C05398=1044.038,401.333,-130.987,174.157,43.481,158.582
C05399=1044.028,401.087,-130.943,174.149,43.474,158.580
C05400=1044.019,400.841,-130.899,174.141,43.469,158.577
C05401=1044.010,400.596,-130.855,174.132,43.462,158.575
C05402=1044.002,400.349,-130.810,174.123,43.456,158.573
C05403=1043.992,400.103,-130.766,174.116,43.450,158.571
C05404=1043.983,399.857,-130.722,174.107,43.444,158.568
C05405=1043.974,399.612,-130.678,174.099,43.437,158.566
C05406=1043.964,399.366,-130.634,174.090,43.432,158.564
C05407=1043.955,399.121,-130.591,174.082,43.426,158.562
C05408=1043.946,398.874,-130.547,174.073,43.420,158.559
C05409=1043.937,398.628,-130.504,174.065,43.414,158.557
C05410=1043.928,398.382,-130.460,174.056,43.408,158.555
C05411=1043.918,398.136,-130.416,174.049,43.402,158.553
C05412=1043.909,397.891,-130.372,174.040,43.396,158.551
C05413=1043.900,397.644,-130.328,174.032,43.390,158.548
C05414=1043.891,397.398,-130.285,174.023,43.384,158.546
C05415=1043.883,397.153,-130.241,174.015,43.378,158.544
C05416=1043.874,396.906,-130.198,174.008,43.372,158.542
C05417=1043.865,396.661,-130.154,173.999,43.366,158.540
C05418=1043.855,396.415,-130.110,173.991,43.360,158.538
C05419=1043.847,396.169,-130.067,173.982,43.355,158.535
C05420=1043.838,395.923,-130.023,173.975,43.349,158.533
C05421=1043.829,395.676,-129.980,173.967,43.343,158.531
C05422=1043.820,395.431,-129.937,173.958,43.337,158.529
C05423=1043.811,395.185,-129.893,173.950,43.331,158.527
C05424=1043.802,394.938,-129.850,173.943,43.325,158.525
C05425=1043.793,394.692,-129.807,173.934,43.320,158.523
C05426=1043.784,394.447,-129.764,173.926,43.314,158.521
C05427=1043.775,394.201,-129.721,173.919,43.308,158.519
C05428=1043.766,393.955,-129.677,173.911,43.303,158.517
C05429=1043.757,393.709,-129.635,173.902,43.297,158.514
C05430=1043.748,393.463,-129.592,173.895,43.291,158.512
C05431=1043.740,393.217,-129.549,173.887,43.286,158.510
C05432=1043.730,392.971,-129.505,173.879,43.280,158.508
C05433=1043.721,392.725,-129.462,173.871,43.275,158.506
C05434=1043.713,392.479,-129.419,173.863,43.269,158.504
C05435=1043.704,392.233,-129.376,173.856,43.264,158.502
C05436=1043.696,391.987,-129.333,173.848,43.258,158.500
C05437=1043.687,391.740,-129.292,173.840,43.252,158.498
C05438=1043.673,391.345,-129.222,173.827,43.244,158.495
C05439=1043.659,390.950,-129.154,173.815,43.235,158.492
C05440=1043.645,390.554,-129.086,173.803,43.226,158.489
C05441=1043.631,390.159,-129.017,173.791,43.217,158.485
C05442=1043.622,389.913,-128.974,173.784,43.212,158.483
C05443=1043.613,389.666,-128.933,173.775,43.206,158.481
C05444=1043.605,389.420,-128.890,173.768,43.201,158.479
C05445=1043.595,389.174,-128.847,173.760,43.196,158.478
C05446=1043.587,388.928,-128.805,173.753,43.190,158.476
C05447=1043.578,388.682,-128.762,173.745,43.185,158.474
C05448=1043.570,388.435,-128.720,173.738,43.179,158.472
C05449=1043.561,388.189,-128.678,173.730,43.174,158.470
C05450=1043.552,387.943,-128.635,173.723,43.169,158.468
C05451=1043.543,387.696,-128.594,173.716,43.164,158.466
C05452=1043.534,387.450,-128.552,173.708,43.158,158.464
C05453=1043.526,387.204,-128.510,173.701,43.153,158.462
C05454=1043.517,386.958,-128.467,173.693,43.148,158.460
C05455=1043.509,386.712,-128.426,173.686,43.143,158.458
C05456=1043.500,386.466,-128.384,173.679,43.137,158.457
C05457=1043.492,386.219,-128.342,173.671,43.133,158.455
C05458=1043.483,385.973,-128.300,173.664,43.127,158.453
C05459=1043.474,385.726,-128.258,173.657,43.122,158.451
C05460=1043.465,385.481,-128.217,173.649,43.117,158.449
C05461=1043.457,385.234,-128.175,173.642,43.112,158.447
C05462=1043.448,384.988,-128.133,173.634,43.107,158.445
C05463=1043.439,384.741,-128.091,173.627,43.102,158.444
C05464=1043.432,384.495,-128.049,173.621,43.097,158.442
C05465=1043.423,384.249,-128.008,173.614,43.091,158.440
C05466=1043.414,384.003,-127.966,173.606,43.086,158.438
C05467=1043.406,383.757,-127.924,173.599,43.082,158.436
C05468=1043.397,383.510,-127.882,173.592,43.077,158.435
C05469=1043.389,383.263,-127.841,173.584,43.071,158.433
C05470=1043.380,383.018,-127.800,173.577,43.066,158.431
C05471=1043.371,382.771,-127.758,173.571,43.061,158.429
C05472=1043.363,382.524,-127.716,173.564,43.056,158.427
C05473=1043.355,382.278,-127.675,173.557,43.052,158.426
C05474=1043.346,382.032,-127.633,173.549,43.047,158.424
C05475=1043.338,381.786,-127.593,173.542,43.042,158.422
C05476=1043.330,381.539,-127.550,173.536,43.037,158.420
C05477=1043.322,381.293,-127.509,173.529,43.032,158.419
C05478=1043.313,381.046,-127.468,173.521,43.027,158.417
C05479=1043.305,380.801,-127.427,173.514,43.022,158.415
C05480=1043.297,380.553,-127.385,173.507,43.017,158.413
C05481=1043.289,380.308,-127.344,173.501,43.012,158.412
C05482=1043.280,380.061,-127.303,173.494,43.007,158.410
C05483=1043.272,379.814,-127.262,173.486,43.002,158.408
C05484=1043.264,379.569,-127.221,173.480,42.997,158.406
C05485=1043.256,379.321,-127.179,173.473,42.992,158.405
C05486=1043.248,379.075,-127.139,173.466,42.988,158.403
C05487=1043.239,378.829,-127.097,173.460,42.983,158.401
C05488=1043.231,378.582,-127.056,173.453,42.978,158.400
C05489=1043.223,378.336,-127.016,173.446,42.974,158.398
C05490=1043.214,378.089,-126.975,173.438,42.969,158.396
C05491=1043.205,377.843,-126.935,173.432,42.964,158.395
C05492=1043.197,377.596,-126.894,173.425,42.959,158.393
C05493=1043.189,377.350,-126.853,173.418,42.955,158.391
C05494=1043.176,376.988,-126.793,173.409,42.948,158.389
C05495=1043.165,376.627,-126.733,173.399,42.941,158.386
C05496=1043.153,376.264,-126.674,173.389,42.934,158.384
C05497=1043.140,375.903,-126.614,173.379,42.928,158.382
C05498=1043.132,375.656,-126.574,173.373,42.923,158.380
C05499=1043.124,375.410,-126.533,173.366,42.919,158.378
C05500=1043.116,375.163,-126.493,173.360,42.914,158.377
C05501=1043.107,374.916,-126.452,173.353,42.909,158.375
C05502=1043.099,374.670,-126.411,173.346,42.905,158.373
C05503=1043.092,374.423,-126.371,173.340,42.900,158.372
C05504=1043.083,374.177,-126.331,173.333,42.896,158.370
C05505=1043.075,373.931,-126.290,173.327,42.891,158.369
C05506=1043.067,373.684,-126.251,173.320,42.887,158.367
C05507=1043.058,373.437,-126.210,173.314,42.882,158.365
C05508=1043.051,373.190,-126.170,173.307,42.877,158.364
C05509=1043.043,372.944,-126.129,173.301,42.873,158.362
C05510=1043.035,372.697,-126.088,173.294,42.869,158.361
C05511=1043.026,372.451,-126.049,173.288,42.864,158.359
C05512=1043.018,372.205,-126.008,173.281,42.860,158.358
C05513=1043.010,371.958,-125.968,173.275,42.855,158.356
C05514=1043.003,371.711,-125.929,173.268,42.851,158.354
C05515=1042.995,371.465,-125.888,173.262,42.846,158.353
C05516=1042.987,371.218,-125.848,173.257,42.842,158.351
C05517=1042.978,370.972,-125.808,173.250,42.838,158.350
C05518=1042.971,370.725,-125.768,173.244,42.833,158.348
C05519=1042.963,370.478,-125.728,173.237,42.829,158.347
C05520=1042.954,370.231,-125.689,173.231,42.824,158.345
C05521=1042.947,369.984,-125.649,173.224,42.821,158.344
C05522=1042.939,369.738,-125.608,173.218,42.816,158.342
C05523=1042.930,369.491,-125.569,173.212,42.812,158.341
C05524=1042.922,369.245,-125.529,173.205,42.808,158.339
C05525=1042.914,368.998,-125.490,173.199,42.803,158.338
C05526=1042.906,368.751,-125.450,173.193,42.799,158.336
C05527=1042.898,368.504,-125.410,173.187,42.795,158.335
C05528=1042.890,368.258,-125.371,173.181,42.791,158.333
C05529=1042.882,368.011,-125.331,173.174,42.786,158.332
C05530=1042.874,367.764,-125.291,173.168,42.782,158.330
C05531=1042.866,367.518,-125.252,173.162,42.778,158.329
C05532=1042.858,367.271,-125.212,173.156,42.774,158.327
C05533=1042.850,367.024,-125.174,173.150,42.769,158.326
C05534=1042.842,366.777,-125.134,173.143,42.766,158.325
C05535=1042.834,366.531,-125.095,173.137,42.762,158.323
C05536=1042.826,366.284,-125.055,173.131,42.757,158.322
C05537=1042.818,366.038,-125.016,173.126,42.753,158.320
C05538=1042.811,365.790,-124.976,173.119,42.749,158.319
C05539=1042.803,365.544,-124.937,173.113,42.745,158.317
C05540=1042.795,365.297,-124.897,173.107,42.741,158.316
C05541=1042.787,365.051,-124.858,173.101,42.737,158.314
C05542=1042.780,364.803,-124.819,173.095,42.732,158.313
C05543=1042.771,364.557,-124.780,173.089,42.728,158.312
C05544=1042.764,364.310,-124.741,173.083,42.724,158.310
C05545=1042.756,364.063,-124.702,173.077,42.721,158.309
C05546=1042.748,363.816,-124.662,173.071,42.717,158.307
C05547=1042.741,363.570,-124.623,173.065,42.713,158.306
C05548=1042.733,363.323,-124.584,173.059,42.708,158.304
C05549=1042.725,363.076,-124.545,173.054,42.704,158.303
C05550=1042.714,362.733,-124.491,173.045,42.698,158.301
C05551=1042.704,362.392,-124.436,173.037,42.693,158.299
C05552=1042.693,362.050,-124.383,173.029,42.688,158.297
C05553=1042.682,361.707,-124.329,173.020,42.682,158.295
C05554=1042.674,361.461,-124.291,173.014,42.678,158.294
C05555=1042.666,361.214,-124.251,173.009,42.674,158.293
C05556=1042.658,360.967,-124.213,173.003,42.670,158.291
C05557=1042.651,360.720,-124.174,172.998,42.667,158.290
C05558=1042.643,360.473,-124.135,172.992,42.663,158.289
C05559=1042.635,360.226,-124.097,172.985,42.659,158.287
C05560=1042.627,359.979,-124.058,172.979,42.655,158.286
C05561=1042.619,359.733,-124.019,172.974,42.651,158.285
C05562=1042.612,359.486,-123.980,172.968,42.647,158.283
C05563=1042.604,359.239,-123.942,172.963,42.643,158.282
C05564=1042.596,358.992,-123.903,172.957,42.639,158.281
C05565=1042.588,358.745,-123.865,172.951,42.636,158.279
C05566=1042.580,358.498,-123.826,172.946,42.632,158.278
C05567=1042.573,358.252,-123.788,172.939,42.628,158.277
C05568=1042.565,358.004,-123.750,172.934,42.625,158.275
C05569=1042.558,357.757,-123.711,172.928,42.621,158.274
C05570=1042.550,357.510,-123.673,172.922,42.617,158.273
C05571=1042.542,357.263,-123.635,172.917,42.613,158.271
C05572=1042.535,357.017,-123.596,172.911,42.610,158.270
C05573=1042.527,356.770,-123.558,172.906,42.606,158.269
C05574=1042.519,356.523,-123.520,172.900,42.602,158.268
C05575=1042.511,356.275,-123.482,172.894,42.598,158.266
C05576=1042.504,356.029,-123.443,172.889,42.595,158.265
C05577=1042.496,355.782,-123.405,172.883,42.591,158.264
C05578=1042.488,355.534,-123.367,172.878,42.587,158.262
C05579=1042.481,355.288,-123.329,172.872,42.584,158.261
C05580=1042.473,355.041,-123.291,172.867,42.580,158.260
C05581=1042.465,354.793,-123.253,172.861,42.576,158.259
C05582=1042.458,354.547,-123.215,172.856,42.573,158.257
C05583=1042.451,354.300,-123.177,172.850,42.569,158.256
C05584=1042.442,354.053,-123.139,172.844,42.565,158.255
C05585=1042.435,353.805,-123.101,172.839,42.562,158.254
C05586=1042.428,353.559,-123.063,172.834,42.558,158.252
C05587=1042.420,353.312,-123.026,172.828,42.555,158.251
C05588=1042.412,353.065,-122.987,172.822,42.551,158.250
C05589=1042.404,352.818,-122.950,172.817,42.547,158.249
C05590=1042.397,352.571,-122.912,172.811,42.544,158.247
C05591=1042.390,352.324,-122.874,172.806,42.540,158.246
C05592=1042.382,352.077,-122.836,172.801,42.537,158.245
C05593=1042.374,351.829,-122.798,172.795,42.533,158.244
C05594=1042.367,351.583,-122.760,172.789,42.529,158.242
C05595=1042.360,351.335,-122.723,172.784,42.526,158.241
C05596=1042.352,351.088,-122.685,172.778,42.522,158.240
C05597=1042.345,350.842,-122.647,172.773,42.519,158.239
C05598=1042.337,350.595,-122.610,172.769,42.515,158.238
C05599=1042.330,350.348,-122.572,172.763,42.512,158.236
C05600=1042.322,350.100,-122.535,172.758,42.508,158.235
C05601=1042.315,349.853,-122.497,172.752,42.505,158.234
C05602=1042.307,349.606,-122.460,172.747,42.501,158.233
C05603=1042.299,349.359,-122.423,172.741,42.498,158.232
C05604=1042.292,349.112,-122.385,172.736,42.495,158.231
C05605=1042.285,348.865,-122.348,172.730,42.492,158.229
C05606=1042.274,348.529,-122.297,172.723,42.486,158.228
C05607=1042.264,348.192,-122.246,172.717,42.482,158.226
C05608=1042.254,347.857,-122.195,172.710,42.477,158.225
C05609=1042.243,347.519,-122.144,172.702,42.473,158.223
C05610=1042.236,347.272,-122.107,172.697,42.469,158.222
C05611=1042.228,347.025,-122.070,172.692,42.466,158.221
C05612=1042.221,346.778,-122.032,172.687,42.463,158.220
C05613=1042.214,346.530,-121.995,172.681,42.460,158.218
C05614=1042.206,346.284,-121.959,172.676,42.456,158.217
C05615=1042.199,346.037,-121.921,172.671,42.452,158.216
C05616=1042.191,345.790,-121.884,172.666,42.450,158.215
C05617=1042.184,345.543,-121.847,172.661,42.446,158.214
C05618=1042.177,345.295,-121.810,172.655,42.443,158.213
C05619=1042.169,345.049,-121.773,172.650,42.440,158.212
C05620=1042.162,344.802,-121.736,172.645,42.436,158.210
C05621=1042.154,344.554,-121.699,172.640,42.433,158.209
C05622=1042.147,344.307,-121.662,172.635,42.430,158.208
C05623=1042.139,344.059,-121.626,172.629,42.427,158.207
C05624=1042.132,343.812,-121.588,172.625,42.423,158.206
C05625=1042.125,343.565,-121.551,172.620,42.420,158.205
C05626=1042.118,343.318,-121.515,172.614,42.417,158.204
C05627=1042.110,343.071,-121.477,172.609,42.414,158.203
C05628=1042.103,342.824,-121.441,172.605,42.410,158.201
C05629=1042.096,342.576,-121.404,172.599,42.407,158.200
C05630=1042.088,342.329,-121.367,172.594,42.404,158.199
C05631=1042.082,342.082,-121.331,172.590,42.401,158.198
C05632=1042.074,341.835,-121.294,172.585,42.398,158.197
C05633=1042.067,341.588,-121.257,172.579,42.394,158.196
C05634=1042.059,341.340,-121.221,172.574,42.391,158.195
C05635=1042.051,341.093,-121.184,172.570,42.388,158.194
C05636=1042.044,340.846,-121.147,172.564,42.385,158.193
C05637=1042.037,340.599,-121.111,172.559,42.382,158.192
C05638=1042.029,340.351,-121.075,172.555,42.379,158.191
C05639=1042.021,340.105,-121.038,172.549,42.376,158.190
C05640=1042.014,339.857,-121.001,172.544,42.372,158.188
C05641=1042.007,339.610,-120.965,172.540,42.369,158.187
C05642=1042.000,339.363,-120.929,172.535,42.366,158.186
C05643=1041.993,339.115,-120.892,172.529,42.363,158.185
C05644=1041.986,338.868,-120.857,172.525,42.360,158.184
C05645=1041.978,338.621,-120.820,172.520,42.357,158.183
C05646=1041.970,338.374,-120.783,172.514,42.354,158.182
C05647=1041.964,338.127,-120.747,172.510,42.351,158.181
C05648=1041.956,337.879,-120.711,172.505,42.348,158.180
C05649=1041.948,337.632,-120.675,172.500,42.345,158.179
C05650=1041.942,337.385,-120.638,172.495,42.342,158.178
C05651=1041.934,337.137,-120.602,172.490,42.339,158.177
C05652=1041.927,336.890,-120.566,172.486,42.336,158.176
C05653=1041.919,336.643,-120.530,172.481,42.333,158.175
C05654=1041.913,336.396,-120.493,172.476,42.330,158.174
C05655=1041.906,336.148,-120.458,172.471,42.327,158.173
C05656=1041.898,335.901,-120.422,172.466,42.324,158.172
C05657=1041.890,335.653,-120.385,172.462,42.321,158.171
C05658=1041.884,335.406,-120.349,172.457,42.318,158.170
C05659=1041.876,335.159,-120.313,172.452,42.315,158.169
C05660=1041.869,334.912,-120.277,172.447,42.312,158.168
C05661=1041.862,334.664,-120.241,172.442,42.309,158.167
C05662=1041.852,334.324,-120.192,172.435,42.305,158.165
C05663=1041.842,333.984,-120.143,172.430,42.301,158.164
C05664=1041.832,333.644,-120.094,172.423,42.297,158.163
C05665=1041.822,333.304,-120.044,172.416,42.293,158.161
C05666=1041.815,333.057,-120.009,172.411,42.290,158.160
C05667=1041.808,332.809,-119.973,172.407,42.287,158.159
C05668=1041.800,332.563,-119.937,172.402,42.284,158.158
C05669=1041.793,332.315,-119.902,172.398,42.281,158.157
C05670=1041.786,332.068,-119.866,172.393,42.278,158.156
C05671=1041.778,331.820,-119.830,172.388,42.275,158.155
C05672=1041.772,331.573,-119.795,172.383,42.273,158.154
C05673=1041.764,331.325,-119.759,172.379,42.270,158.153
C05674=1041.757,331.078,-119.723,172.374,42.267,158.152
C05675=1041.750,330.831,-119.688,172.370,42.264,158.152
C05676=1041.743,330.583,-119.652,172.365,42.261,158.151
C05677=1041.736,330.336,-119.617,172.360,42.258,158.150
C05678=1041.728,330.089,-119.580,172.355,42.256,158.149
C05679=1041.722,329.841,-119.545,172.351,42.253,158.148
C05680=1041.715,329.594,-119.510,172.346,42.250,158.147
C05681=1041.707,329.346,-119.474,172.342,42.247,158.146
C05682=1041.700,329.099,-119.439,172.338,42.244,158.145
C05683=1041.693,328.852,-119.404,172.333,42.241,158.144
C05684=1041.685,328.604,-119.369,172.328,42.239,158.143
C05685=1041.678,328.357,-119.333,172.323,42.236,158.142
C05686=1041.670,328.109,-119.298,172.319,42.233,158.141
C05687=1041.663,327.862,-119.263,172.314,42.231,158.140
C05688=1041.656,327.615,-119.228,172.310,42.228,158.139
C05689=1041.649,327.367,-119.193,172.305,42.225,158.138
C05690=1041.642,327.120,-119.158,172.301,42.223,158.137
C05691=1041.634,326.873,-119.123,172.296,42.220,158.136
C05692=1041.627,326.624,-119.088,172.292,42.217,158.136
C05693=1041.619,326.377,-119.053,172.287,42.215,158.135
C05694=1041.613,326.130,-119.018,172.283,42.212,158.134
C05695=1041.605,325.882,-118.983,172.279,42.209,158.133
C05696=1041.598,325.635,-118.948,172.274,42.207,158.132
C05697=1041.591,325.388,-118.913,172.269,42.204,158.131
C05698=1041.584,325.140,-118.878,172.264,42.201,158.130
C05699=1041.576,324.892,-118.843,172.260,42.199,158.129
C05700=1041.569,324.645,-118.808,172.256,42.196,158.128
C05701=1041.562,324.398,-118.773,172.251,42.193,158.127
C05702=1041.554,324.151,-118.739,172.247,42.191,158.127
C05703=1041.548,323.903,-118.704,172.242,42.188,158.126
C05704=1041.541,323.655,-118.669,172.238,42.185,158.125
C05705=1041.533,323.408,-118.634,172.234,42.183,158.124
C05706=1041.526,323.160,-118.599,172.229,42.180,158.123
C05707=1041.519,322.913,-118.564,172.225,42.178,158.122
C05708=1041.512,322.665,-118.530,172.221,42.175,158.121
C05709=1041.505,322.418,-118.496,172.216,42.172,158.120
C05710=1041.497,322.170,-118.460,172.212,42.170,158.119
C05711=1041.490,321.923,-118.425,172.208,42.167,158.119
C05712=1041.483,321.675,-118.391,172.203,42.165,158.118
C05713=1041.476,321.428,-118.357,172.199,42.162,158.117
C05714=1041.469,321.181,-118.321,172.195,42.160,158.116
C05715=1041.462,320.933,-118.288,172.189,42.157,158.115
C05716=1041.455,320.686,-118.252,172.185,42.154,158.114
C05717=1041.448,320.438,-118.219,172.181,42.152,158.113
C05718=1041.438,320.094,-118.169,172.175,42.148,158.112
C05719=1041.428,319.749,-118.121,172.170,42.145,158.111
C05720=1041.418,319.404,-118.073,172.163,42.141,158.110
C05721=1041.409,319.059,-118.025,172.157,42.138,158.108
C05722=1041.402,318.811,-117.991,172.153,42.135,158.108
C05723=1041.395,318.564,-117.956,172.149,42.133,158.107
C05724=1041.388,318.316,-117.922,172.145,42.130,158.106
C05725=1041.381,318.069,-117.887,172.140,42.128,158.105
C05726=1041.375,317.822,-117.854,172.136,42.125,158.104
C05727=1041.368,317.574,-117.818,172.132,42.123,158.103
C05728=1041.361,317.327,-117.785,172.128,42.120,158.103
C05729=1041.353,317.079,-117.751,172.123,42.118,158.102
C05730=1041.347,316.832,-117.716,172.119,42.115,158.101
C05731=1041.339,316.584,-117.682,172.115,42.113,158.100
C05732=1041.333,316.337,-117.647,172.111,42.110,158.099
C05733=1041.326,316.089,-117.613,172.107,42.108,158.098
C05734=1041.319,315.841,-117.578,172.102,42.105,158.097
C05735=1041.312,315.593,-117.545,172.098,42.103,158.097
C05736=1041.306,315.347,-117.510,172.094,42.100,158.096
C05737=1041.298,315.099,-117.476,172.090,42.098,158.095
C05738=1041.292,314.851,-117.442,172.086,42.095,158.094
C05739=1041.285,314.604,-117.407,172.081,42.093,158.093
C05740=1041.278,314.356,-117.373,172.077,42.090,158.092
C05741=1041.271,314.109,-117.339,172.073,42.088,158.092
C05742=1041.265,313.861,-117.305,172.069,42.085,158.091
C05743=1041.258,313.613,-117.271,172.065,42.083,158.090
C05744=1041.251,313.366,-117.237,172.061,42.080,158.089
C05745=1041.244,313.119,-117.202,172.056,42.078,158.088
C05746=1041.237,312.871,-117.169,172.052,42.075,158.087
C05747=1041.231,312.623,-117.134,172.048,42.073,158.087
C05748=1041.224,312.376,-117.100,172.044,42.070,158.086
C05749=1041.217,312.129,-117.067,172.040,42.068,158.085
C05750=1041.210,311.881,-117.033,172.036,42.066,158.084
C05751=1041.203,311.633,-116.999,172.031,42.063,158.083
C05752=1041.195,311.386,-116.965,172.027,42.062,158.083
C05753=1041.188,311.138,-116.932,172.023,42.059,158.082
C05754=1041.181,310.890,-116.898,172.020,42.057,158.081
C05755=1041.175,310.643,-116.865,172.016,42.054,158.080
C05756=1041.167,310.395,-116.831,172.012,42.052,158.080
C05757=1041.160,310.147,-116.797,172.007,42.050,158.079
C05758=1041.150,309.818,-116.753,172.002,42.047,158.078
C05759=1041.141,309.488,-116.708,171.997,42.044,158.077
C05760=1041.131,309.159,-116.664,171.991,42.041,158.076
C05761=1041.123,308.829,-116.620,171.986,42.038,158.075
C05762=1041.116,308.581,-116.586,171.982,42.035,158.074
C05763=1041.108,308.334,-116.552,171.977,42.034,158.073
C05764=1041.102,308.086,-116.520,171.973,42.031,158.072
C05765=1041.095,307.838,-116.486,171.970,42.029,158.072
C05766=1041.087,307.591,-116.453,171.966,42.027,158.071
C05767=1041.080,307.343,-116.419,171.962,42.025,158.070
C05768=1041.073,307.096,-116.386,171.958,42.022,158.069
C05769=1041.066,306.848,-116.352,171.954,42.020,158.069
C05770=1041.060,306.600,-116.319,171.950,42.018,158.068
C05771=1041.053,306.353,-116.286,171.946,42.015,158.067
C05772=1041.045,306.105,-116.253,171.941,42.014,158.066
C05773=1041.038,305.858,-116.220,171.937,42.011,158.066
C05774=1041.031,305.599,-116.185,171.934,42.009,158.065
C05775=1041.024,305.341,-116.150,171.930,42.007,158.064
C05776=1041.017,305.084,-116.116,171.926,42.004,158.063
C05777=1041.010,304.825,-116.081,171.922,42.002,158.063
C05778=1041.003,304.578,-116.048,171.918,42.000,158.062
C05779=1040.996,304.330,-116.015,171.914,41.997,158.061
C05780=1040.990,304.082,-115.982,171.909,41.996,158.060
C05781=1040.982,303.835,-115.949,171.905,41.993,158.059
C05782=1040.976,303.587,-115.916,171.902,41.991,158.059
C05783=1040.968,303.340,-115.882,171.898,41.989,158.058
C05784=1040.961,303.091,-115.849,171.894,41.987,158.057
C05785=1040.955,302.844,-115.816,171.890,41.985,158.057
C05786=1040.948,302.597,-115.783,171.886,41.983,158.056
C05787=1040.941,302.349,-115.750,171.882,41.980,158.055
C05788=1040.935,302.101,-115.718,171.878,41.978,158.054
C05789=1040.927,301.854,-115.684,171.875,41.976,158.054
C05790=1040.921,301.606,-115.651,171.871,41.974,158.053
C05791=1040.914,301.358,-115.618,171.867,41.972,158.052
C05792=1040.907,301.110,-115.586,171.863,41.970,158.051
C05793=1040.900,300.863,-115.552,171.859,41.967,158.051
C05794=1040.894,300.615,-115.519,171.855,41.965,158.050
C05795=1040.887,300.367,-115.486,171.852,41.963,158.049
C05796=1040.880,300.120,-115.454,171.849,41.960,158.048
C05797=1040.873,299.872,-115.421,171.845,41.958,158.048
C05798=1040.866,299.624,-115.387,171.841,41.956,158.047
C05799=1040.860,299.377,-115.355,171.837,41.954,158.046
C05800=1040.854,299.129,-115.322,171.833,41.952,158.046
C05801=1040.846,298.881,-115.289,171.829,41.950,158.045
C05802=1040.840,298.634,-115.257,171.826,41.948,158.044
C05803=1040.833,298.386,-115.224,171.822,41.946,158.044
C05804=1040.827,298.138,-115.191,171.818,41.943,158.043
C05805=1040.820,297.890,-115.159,171.814,41.941,158.042
C05806=1040.813,297.643,-115.126,171.810,41.939,158.041
C05807=1040.806,297.394,-115.093,171.807,41.937,158.041
C05808=1040.800,297.147,-115.060,171.803,41.935,158.040
C05809=1040.794,296.899,-115.027,171.799,41.933,158.039
C05810=1040.786,296.651,-114.995,171.796,41.931,158.039
C05811=1040.780,296.404,-114.962,171.792,41.929,158.038
C05812=1040.774,296.156,-114.929,171.788,41.927,158.037
C05813=1040.767,295.909,-114.897,171.784,41.924,158.036
C05814=1040.760,295.661,-114.864,171.781,41.922,158.036
C05815=1040.753,295.413,-114.831,171.777,41.920,158.035
C05816=1040.747,295.165,-114.799,171.773,41.918,158.034
C05817=1040.739,294.917,-114.766,171.769,41.916,158.034
C05818=1040.733,294.669,-114.735,171.766,41.914,158.033
C05819=1040.726,294.422,-114.702,171.763,41.912,158.032
C05820=1040.719,294.175,-114.670,171.759,41.910,158.032
C05821=1040.712,293.926,-114.637,171.755,41.908,158.031
C05822=1040.706,293.678,-114.605,171.751,41.906,158.030
C05823=1040.699,293.431,-114.572,171.748,41.904,158.030
C05824=1040.692,293.183,-114.540,171.744,41.902,158.029
C05825=1040.685,292.935,-114.508,171.740,41.900,158.028
C05826=1040.679,292.687,-114.476,171.736,41.898,158.028
C05827=1040.672,292.440,-114.444,171.734,41.896,158.027
C05828=1040.664,292.191,-114.412,171.730,41.894,158.026
C05829=1040.658,291.944,-114.379,171.726,41.892,158.026
C05830=1040.649,291.621,-114.337,171.721,41.889,158.025
C05831=1040.640,291.296,-114.295,171.716,41.887,158.024
C05832=1040.631,290.973,-114.254,171.712,41.884,158.023
C05833=1040.623,290.650,-114.212,171.707,41.882,158.022
C05834=1040.616,290.402,-114.180,171.703,41.880,158.021
C05835=1040.609,290.155,-114.148,171.700,41.878,158.021
C05836=1040.603,289.906,-114.116,171.696,41.876,158.020
C05837=1040.596,289.658,-114.084,171.693,41.874,158.019
C05838=1040.589,289.411,-114.052,171.689,41.872,158.019
C05839=1040.582,289.163,-114.020,171.685,41.870,158.018
C05840=1040.575,288.915,-113.987,171.682,41.868,158.018
C05841=1040.569,288.667,-113.956,171.678,41.866,158.017
C05842=1040.562,288.419,-113.925,171.675,41.864,158.016
C05843=1040.555,288.172,-113.892,171.672,41.862,158.016
C05844=1040.549,287.924,-113.860,171.668,41.860,158.015
C05845=1040.542,287.676,-113.828,171.664,41.858,158.014
C05846=1040.535,287.428,-113.797,171.660,41.857,158.014
C05847=1040.528,287.180,-113.765,171.658,41.855,158.013
C05848=1040.521,286.932,-113.734,171.654,41.853,158.012
C05849=1040.514,286.685,-113.701,171.650,41.851,158.012
C05850=1040.507,286.437,-113.670,171.646,41.849,158.011
C05851=1040.501,286.189,-113.638,171.643,41.847,158.010
C05852=1040.495,285.941,-113.607,171.640,41.845,158.010
C05853=1040.488,285.693,-113.575,171.636,41.843,158.009
C05854=1040.481,285.446,-113.543,171.633,41.842,158.009
C05855=1040.474,285.198,-113.512,171.629,41.840,158.008
C05856=1040.467,284.949,-113.480,171.626,41.838,158.007
C05857=1040.460,284.701,-113.448,171.622,41.836,158.007
C05858=1040.453,284.453,-113.417,171.619,41.834,158.006
C05859=1040.447,284.205,-113.385,171.615,41.832,158.005
C05860=1040.440,283.957,-113.354,171.612,41.831,158.005
C05861=1040.433,283.709,-113.323,171.609,41.829,158.004
C05862=1040.426,283.462,-113.291,171.605,41.827,158.004
C05863=1040.420,283.214,-113.260,171.601,41.825,158.003
C05864=1040.413,282.966,-113.228,171.598,41.823,158.002
C05865=1040.406,282.718,-113.197,171.595,41.821,158.002
C05866=1040.400,282.470,-113.165,171.591,41.820,158.001
C05867=1040.393,282.222,-113.134,171.587,41.818,158.001
C05868=1040.386,281.974,-113.103,171.585,41.816,158.000
C05869=1040.379,281.726,-113.071,171.581,41.814,157.999
C05870=1040.373,281.478,-113.040,171.577,41.812,157.999
C05871=1040.366,281.230,-113.008,171.574,41.810,157.998
C05872=1040.359,280.983,-112.977,171.571,41.809,157.998
C05873=1040.352,280.735,-112.945,171.567,41.807,157.997
C05874=1040.346,280.487,-112.914,171.564,41.804,157.996
C05875=1040.339,280.239,-112.883,171.561,41.803,157.996
C05876=1040.333,279.991,-112.852,171.557,41.801,157.995
C05877=1040.326,279.743,-112.821,171.553,41.800,157.994
C05878=1040.320,279.495,-112.789,171.551,41.798,157.994
C05879=1040.313,279.247,-112.758,171.547,41.796,157.993
C05880=1040.306,279.000,-112.727,171.543,41.794,157.993
C05881=1040.299,278.752,-112.696,171.540,41.792,157.992
C05882=1040.292,278.503,-112.665,171.537,41.791,157.991
C05883=1040.286,278.255,-112.634,171.533,41.789,157.991
C05884=1040.279,278.007,-112.602,171.531,41.787,157.990
C05885=1040.273,277.759,-112.571,171.527,41.785,157.990
C05886=1040.264,277.448,-112.533,171.523,41.783,157.989
C05887=1040.255,277.136,-112.494,171.518,41.780,157.988
C05888=1040.247,276.825,-112.455,171.514,41.778,157.987
C05889=1040.239,276.513,-112.416,171.510,41.776,157.987
C05890=1040.232,276.265,-112.384,171.507,41.774,157.986
C05891=1040.225,276.017,-112.354,171.504,41.772,157.985
C05892=1040.218,275.769,-112.323,171.500,41.771,157.985
C05893=1040.212,275.521,-112.292,171.497,41.769,157.984
C05894=1040.205,275.273,-112.261,171.494,41.767,157.984
C05895=1040.198,275.025,-112.231,171.490,41.766,157.983
C05896=1040.192,274.777,-112.199,171.487,41.764,157.983
C05897=1040.185,274.529,-112.169,171.484,41.762,157.982
C05898=1040.178,274.281,-112.138,171.480,41.760,157.981
C05899=1040.171,274.033,-112.107,171.478,41.759,157.981
C05900=1040.165,273.785,-112.076,171.474,41.757,157.980
C05901=1040.158,273.537,-112.046,171.470,41.755,157.980
C05902=1040.151,273.289,-112.014,171.468,41.754,157.979
C05903=1040.145,273.041,-111.984,171.464,41.752,157.979
C05904=1040.138,272.793,-111.954,171.462,41.750,157.978
C05905=1040.131,272.545,-111.922,171.458,41.748,157.977
C05906=1040.125,272.297,-111.892,171.454,41.747,157.977
C05907=1040.118,272.049,-111.861,171.451,41.745,157.976
C05908=1040.111,271.801,-111.830,171.448,41.743,157.976
C05909=1040.104,271.553,-111.800,171.445,41.742,157.975
C05910=1040.098,271.305,-111.769,171.442,41.740,157.975
C05911=1040.092,271.057,-111.738,171.438,41.738,157.974
C05912=1040.085,270.809,-111.708,171.435,41.737,157.973
C05913=1040.078,270.560,-111.678,171.432,41.735,157.973
C05914=1040.071,270.313,-111.647,171.429,41.733,157.972
C05915=1040.065,270.065,-111.616,171.425,41.732,157.972
C05916=1040.058,269.816,-111.586,171.423,41.729,157.971
C05917=1040.051,269.568,-111.556,171.419,41.728,157.971
C05918=1040.045,269.320,-111.526,171.417,41.726,157.970
C05919=1040.037,269.073,-111.495,171.413,41.724,157.969
C05920=1040.031,268.824,-111.464,171.409,41.723,157.969
C05921=1040.024,268.577,-111.434,171.407,41.721,157.968
C05922=1040.018,268.328,-111.404,171.403,41.719,157.968
C05923=1040.011,268.080,-111.374,171.400,41.718,157.967
C05924=1040.005,267.832,-111.343,171.397,41.716,157.967
C05925=1039.998,267.584,-111.313,171.394,41.715,157.966
C05926=1039.991,267.335,-111.282,171.390,41.713,157.966
C05927=1039.985,267.089,-111.252,171.388,41.711,157.965
C05928=1039.977,266.840,-111.222,171.384,41.710,157.965
C05929=1039.971,266.592,-111.191,171.382,41.708,157.964
C05930=1039.964,266.344,-111.161,171.378,41.706,157.963
C05931=1039.957,266.096,-111.131,171.375,41.705,157.963
C05932=1039.951,265.848,-111.101,171.372,41.703,157.962
C05933=1039.944,265.600,-111.071,171.369,41.702,157.962
C05934=1039.937,265.351,-111.041,171.365,41.700,157.961
C05935=1039.931,265.103,-111.011,171.363,41.698,157.961
C05936=1039.924,264.855,-110.981,171.359,41.697,157.960
C05937=1039.917,264.607,-110.951,171.357,41.695,157.960
C05938=1039.911,264.358,-110.920,171.353,41.693,157.959
C05939=1039.904,264.111,-110.890,171.350,41.692,157.959
C05940=1039.897,263.863,-110.860,171.347,41.690,157.958
C05941=1039.891,263.615,-110.830,171.344,41.689,157.958
C05942=1039.883,263.308,-110.793,171.340,41.687,157.957
C05943=1039.874,263.000,-110.755,171.337,41.685,157.956
C05944=1039.866,262.693,-110.718,171.333,41.683,157.956
C05945=1039.858,262.386,-110.681,171.329,41.680,157.955
C05946=1039.852,262.138,-110.652,171.326,41.679,157.954
C05947=1039.845,261.890,-110.622,171.323,41.677,157.954
C05948=1039.838,261.642,-110.591,171.319,41.676,157.953
C05949=1039.831,261.394,-110.562,171.317,41.674,157.953
C05950=1039.824,261.146,-110.532,171.313,41.672,157.952
C05951=1039.818,260.898,-110.503,171.311,41.671,157.952
C05952=1039.811,260.649,-110.473,171.307,41.669,157.951
C05953=1039.804,260.401,-110.443,171.304,41.668,157.951
C05954=1039.797,260.153,-110.414,171.301,41.666,157.950
C05955=1039.790,259.905,-110.384,171.298,41.665,157.950
C05956=1039.784,259.657,-110.354,171.295,41.663,157.949
C05957=1039.776,259.409,-110.325,171.292,41.662,157.949
C05958=1039.769,259.161,-110.296,171.289,41.660,157.948
C05959=1039.763,258.912,-110.266,171.286,41.659,157.948
C05960=1039.755,258.664,-110.236,171.283,41.657,157.947
C05961=1039.749,258.416,-110.207,171.280,41.656,157.947
C05962=1039.742,258.168,-110.177,171.277,41.654,157.946
C05963=1039.736,257.920,-110.148,171.274,41.653,157.946
C05964=1039.729,257.671,-110.118,171.271,41.651,157.945
C05965=1039.722,257.423,-110.089,171.268,41.650,157.945
C05966=1039.715,257.175,-110.059,171.265,41.648,157.944
C05967=1039.709,256.927,-110.029,171.262,41.647,157.944
C05968=1039.702,256.679,-109.999,171.259,41.645,157.943
C05969=1039.695,256.431,-109.971,171.256,41.644,157.943
C05970=1039.688,256.182,-109.941,171.253,41.642,157.942
C05971=1039.681,255.934,-109.912,171.250,41.641,157.942
C05972=1039.675,255.686,-109.882,171.248,41.639,157.941
C05973=1039.668,255.438,-109.853,171.244,41.638,157.941
C05974=1039.662,255.190,-109.824,171.242,41.636,157.940
C05975=1039.655,254.941,-109.794,171.238,41.635,157.940
C05976=1039.648,254.694,-109.764,171.235,41.633,157.939
C05977=1039.641,254.445,-109.735,171.233,41.632,157.939
C05978=1039.635,254.197,-109.706,171.229,41.630,157.938
C05979=1039.627,253.949,-109.676,171.227,41.629,157.938
C05980=1039.621,253.701,-109.647,171.224,41.627,157.937
C05981=1039.615,253.453,-109.618,171.221,41.626,157.937
C05982=1039.608,253.204,-109.588,171.218,41.624,157.936
C05983=1039.601,252.956,-109.559,171.215,41.623,157.936
C05984=1039.595,252.707,-109.530,171.212,41.621,157.935
C05985=1039.588,252.459,-109.501,171.209,41.619,157.935
C05986=1039.582,252.212,-109.471,171.207,41.618,157.934
C05987=1039.574,251.963,-109.442,171.203,41.616,157.934
C05988=1039.568,251.715,-109.413,171.201,41.615,157.933
C05989=1039.562,251.467,-109.384,171.198,41.613,157.933
C05990=1039.555,251.218,-109.355,171.194,41.612,157.932
C05991=1039.548,250.971,-109.325,171.192,41.610,157.932
C05992=1039.542,250.722,-109.296,171.189,41.609,157.931
C05993=1039.535,250.474,-109.266,171.186,41.607,157.931
C05994=1039.529,250.225,-109.237,171.183,41.606,157.930
C05995=1039.522,249.978,-109.209,171.181,41.604,157.930
C05996=1039.515,249.729,-109.180,171.177,41.603,157.929
C05997=1039.509,249.481,-109.151,171.175,41.601,157.929
C05998=1039.501,249.172,-109.114,171.171,41.599,157.928
C05999=1039.493,248.864,-109.078,171.167,41.598,157.927
C06000=1039.485,248.556,-109.041,171.164,41.595,157.927
C06001=1039.476,248.247,-109.005,171.161,41.593,157.926
C06002=1039.470,247.999,-108.976,171.158,41.592,157.926
C06003=1039.464,247.751,-108.947,171.155,41.590,157.925
C06004=1039.456,247.502,-108.918,171.152,41.589,157.925
C06005=1039.450,247.254,-108.889,171.149,41.587,157.924
C06006=1039.444,247.006,-108.860,171.147,41.586,157.924
C06007=1039.437,246.758,-108.831,171.143,41.584,157.923
C06008=1039.431,246.509,-108.802,171.141,41.583,157.923
C06009=1039.424,246.261,-108.773,171.138,41.581,157.922
C06010=1039.418,246.013,-108.743,171.136,41.579,157.922
C06011=1039.411,245.765,-108.715,171.132,41.578,157.921
C06012=1039.405,245.517,-108.686,171.130,41.576,157.921
C06013=1039.398,245.268,-108.657,171.127,41.575,157.920
C06014=1039.392,245.019,-108.628,171.124,41.573,157.920
C06015=1039.385,244.771,-108.600,171.121,41.572,157.919
C06016=1039.379,244.523,-108.571,171.118,41.570,157.919
C06017=1039.373,244.275,-108.542,171.116,41.569,157.918
C06018=1039.365,244.027,-108.513,171.113,41.568,157.918
C06019=1039.359,243.778,-108.484,171.110,41.566,157.917
C06020=1039.352,243.530,-108.456,171.107,41.565,157.917
C06021=1039.346,243.282,-108.427,171.105,41.563,157.916
C06022=1039.339,243.034,-108.399,171.102,41.562,157.916
C06023=1039.332,242.785,-108.369,171.100,41.560,157.915
C06024=1039.326,242.536,-108.341,171.096,41.558,157.915
C06025=1039.319,242.289,-108.312,171.093,41.557,157.914
C06026=1039.313,242.040,-108.283,171.091,41.556,157.914
C06027=1039.306,241.793,-108.255,171.088,41.554,157.914
C06028=1039.300,241.544,-108.227,171.086,41.553,157.913
C06029=1039.293,241.295,-108.197,171.082,41.551,157.913
C06030=1039.286,241.047,-108.169,171.080,41.550,157.912
C06031=1039.280,240.799,-108.141,171.077,41.548,157.912
C06032=1039.273,240.551,-108.112,171.075,41.547,157.911
C06033=1039.266,240.302,-108.084,171.072,41.546,157.911
C06034=1039.260,240.054,-108.055,171.069,41.544,157.910
C06035=1039.253,239.806,-108.027,171.066,41.543,157.910
C06036=1039.246,239.557,-107.999,171.064,41.541,157.909
C06037=1039.240,239.309,-107.970,171.061,41.539,157.909
C06038=1039.233,239.061,-107.942,171.059,41.538,157.908
C06039=1039.226,238.813,-107.914,171.055,41.537,157.908
C06040=1039.220,238.564,-107.885,171.053,41.535,157.907
C06041=1039.213,238.316,-107.857,171.050,41.534,157.907
C06042=1039.206,238.068,-107.829,171.048,41.533,157.907
C06043=1039.199,237.819,-107.800,171.045,41.531,157.906
C06044=1039.193,237.570,-107.772,171.042,41.530,157.906
C06045=1039.186,237.323,-107.743,171.039,41.528,157.905
C06046=1039.179,237.074,-107.716,171.037,41.527,157.905
C06047=1039.173,236.825,-107.687,171.034,41.526,157.904
C06048=1039.166,236.578,-107.659,171.031,41.524,157.904
C06049=1039.160,236.329,-107.631,171.029,41.522,157.903
C06050=1039.153,236.081,-107.603,171.026,41.521,157.903
C06051=1039.147,235.833,-107.574,171.023,41.520,157.902
C06052=1039.140,235.584,-107.547,171.020,41.518,157.902
C06053=1039.133,235.336,-107.518,171.018,41.517,157.901
C06054=1039.124,235.022,-107.483,171.014,41.515,157.901
C06055=1039.117,234.707,-107.447,171.012,41.513,157.900
C06056=1039.108,234.393,-107.411,171.008,41.512,157.900
C06057=1039.099,234.078,-107.376,171.004,41.510,157.899
C06058=1039.092,233.830,-107.348,171.002,41.508,157.899
C06059=1039.086,233.582,-107.319,170.999,41.507,157.898
C06060=1039.079,233.333,-107.291,170.997,41.506,157.898
C06061=1039.073,233.085,-107.263,170.994,41.504,157.897
C06062=1039.066,232.836,-107.236,170.992,41.502,157.897
C06063=1039.060,232.588,-107.207,170.989,41.501,157.897
C06064=1039.053,232.340,-107.179,170.987,41.500,157.896
C06065=1039.046,232.091,-107.151,170.984,41.498,157.896
C06066=1039.040,231.843,-107.124,170.981,41.497,157.895
C06067=1039.033,231.595,-107.095,170.978,41.495,157.895
C06068=1039.026,231.347,-107.067,170.976,41.494,157.894
C06069=1039.020,231.098,-107.039,170.973,41.493,157.894
C06070=1039.013,230.849,-107.011,170.971,41.491,157.893
C06071=1039.007,230.601,-106.984,170.968,41.490,157.893
C06072=1039.000,230.353,-106.956,170.966,41.488,157.892
C06073=1038.993,230.104,-106.928,170.963,41.487,157.892
C06074=1038.987,229.856,-106.900,170.961,41.485,157.891
C06075=1038.980,229.608,-106.872,170.958,41.484,157.891
C06076=1038.974,229.360,-106.845,170.956,41.483,157.891
C06077=1038.967,229.112,-106.817,170.953,41.481,157.890
C06078=1038.960,228.863,-106.789,170.950,41.480,157.890
C06079=1038.954,228.615,-106.761,170.947,41.479,157.889
C06080=1038.948,228.366,-106.733,170.945,41.477,157.889
C06081=1038.940,228.118,-106.706,170.942,41.475,157.888
C06082=1038.934,227.870,-106.678,170.940,41.474,157.888
C06083=1038.927,227.621,-106.650,170.937,41.473,157.887
C06084=1038.920,227.373,-106.623,170.935,41.472,157.887
C06085=1038.914,227.124,-106.595,170.932,41.470,157.887
C06086=1038.907,226.876,-106.567,170.930,41.469,157.886
C06087=1038.900,226.627,-106.540,170.927,41.468,157.886
C06088=1038.894,226.378,-106.513,170.925,41.466,157.885
C06089=1038.886,226.130,-106.485,170.922,41.465,157.885
C06090=1038.880,225.882,-106.458,170.920,41.464,157.885
C06091=1038.873,225.633,-106.430,170.917,41.462,157.884
C06092=1038.867,225.386,-106.403,170.915,41.460,157.884
C06093=1038.860,225.137,-106.375,170.912,41.459,157.883
C06094=1038.854,224.889,-106.347,170.910,41.458,157.883
C06095=1038.847,224.640,-106.319,170.907,41.456,157.882
C06096=1038.840,224.391,-106.293,170.905,41.455,157.882
C06097=1038.833,224.143,-106.265,170.902,41.454,157.881
C06098=1038.826,223.895,-106.237,170.900,41.453,157.881
C06099=1038.820,223.646,-106.210,170.897,41.451,157.881
C06100=1038.814,223.398,-106.182,170.895,41.449,157.880
C06101=1038.807,223.149,-106.155,170.892,41.448,157.880
C06102=1038.800,222.901,-106.128,170.890,41.447,157.879
C06103=1038.793,222.653,-106.100,170.887,41.445,157.879
C06104=1038.787,222.404,-106.073,170.885,41.444,157.878
C06105=1038.780,222.155,-106.046,170.882,41.443,157.878
C06106=1038.774,221.907,-106.018,170.880,41.441,157.878
C06107=1038.767,221.659,-105.991,170.878,41.440,157.877
C06108=1038.760,221.411,-105.964,170.875,41.438,157.877
C06109=1038.754,221.162,-105.937,170.872,41.437,157.876
C06110=1038.746,220.840,-105.901,170.869,41.435,157.876
C06111=1038.737,220.518,-105.866,170.866,41.433,157.875
C06112=1038.728,220.197,-105.831,170.863,41.432,157.875
C06113=1038.720,219.875,-105.795,170.860,41.429,157.874
C06114=1038.713,219.627,-105.768,170.857,41.428,157.874
C06115=1038.706,219.378,-105.741,170.855,41.427,157.873
C06116=1038.699,219.129,-105.714,170.853,41.426,157.873
C06117=1038.692,218.881,-105.686,170.850,41.424,157.872
C06118=1038.686,218.632,-105.659,170.848,41.423,157.872
C06119=1038.679,218.385,-105.632,170.845,41.422,157.871
C06120=1038.673,218.135,-105.605,170.843,41.420,157.871
C06121=1038.665,217.887,-105.578,170.840,41.419,157.871
C06122=1038.659,217.638,-105.551,170.838,41.418,157.870
C06123=1038.652,217.391,-105.524,170.835,41.417,157.870
C06124=1038.646,217.142,-105.497,170.833,41.415,157.869
C06125=1038.639,216.893,-105.469,170.830,41.414,157.869
C06126=1038.632,216.645,-105.443,170.828,41.412,157.869
C06127=1038.625,216.396,-105.415,170.825,41.411,157.868
C06128=1038.619,216.148,-105.389,170.823,41.410,157.868
C06129=1038.612,215.899,-105.362,170.820,41.408,157.867
C06130=1038.605,215.651,-105.335,170.818,41.407,157.867
C06131=1038.599,215.403,-105.308,170.815,41.406,157.866
C06132=1038.592,215.154,-105.281,170.814,41.404,157.866
C06133=1038.585,214.905,-105.254,170.812,41.403,157.866
C06134=1038.578,214.657,-105.227,170.809,41.401,157.865
C06135=1038.572,214.409,-105.200,170.807,41.400,157.865
C06136=1038.566,214.160,-105.173,170.804,41.399,157.864
C06137=1038.558,213.912,-105.146,170.802,41.397,157.864
C06138=1038.553,213.663,-105.120,170.799,41.396,157.863
C06139=1038.546,213.415,-105.093,170.797,41.394,157.863
C06140=1038.539,213.166,-105.065,170.794,41.393,157.863
C06141=1038.532,212.918,-105.039,170.793,41.392,157.862
C06142=1038.526,212.669,-105.012,170.790,41.390,157.862
C06143=1038.519,212.421,-104.985,170.788,41.389,157.861
C06144=1038.513,212.173,-104.959,170.785,41.388,157.861
C06145=1038.506,211.924,-104.932,170.783,41.386,157.860
C06146=1038.499,211.675,-104.904,170.780,41.385,157.860
C06147=1038.492,211.427,-104.878,170.778,41.383,157.860
C06148=1038.486,211.178,-104.851,170.775,41.382,157.859
C06149=1038.479,210.929,-104.825,170.774,41.381,157.859
C06150=1038.473,210.682,-104.798,170.772,41.380,157.858
C06151=1038.466,210.433,-104.771,170.769,41.378,157.858
C06152=1038.459,210.184,-104.745,170.766,41.376,157.858
C06153=1038.453,209.936,-104.718,170.764,41.375,157.857
C06154=1038.446,209.687,-104.692,170.762,41.374,157.857
C06155=1038.439,209.439,-104.666,170.759,41.373,157.856
C06156=1038.433,209.191,-104.638,170.758,41.371,157.856
C06157=1038.426,208.942,-104.612,170.755,41.370,157.856
C06158=1038.419,208.694,-104.585,170.753,41.368,157.855
C06159=1038.413,208.445,-104.558,170.750,41.367,157.855
C06160=1038.406,208.196,-104.532,170.748,41.366,157.854
C06161=1038.399,207.948,-104.506,170.745,41.364,157.854
C06162=1038.392,207.699,-104.480,170.743,41.363,157.853
C06163=1038.386,207.451,-104.453,170.741,41.361,157.853
C06164=1038.379,207.202,-104.426,170.739,41.361,157.853
C06165=1038.372,206.953,-104.400,170.736,41.359,157.852
C06166=1038.364,206.638,-104.366,170.734,41.357,157.852
C06167=1038.355,206.321,-104.333,170.730,41.356,157.851
C06168=1038.347,206.005,-104.299,170.728,41.354,157.851
C06169=1038.338,205.689,-104.266,170.725,41.352,157.850
C06170=1038.312,204.638,-104.159,170.425,41.248,157.812
C06171=1038.306,204.390,-104.134,170.421,41.248,157.812
C06172=1038.300,204.141,-104.109,170.418,41.247,157.811
C06173=1038.293,203.893,-104.084,170.415,41.247,157.811
C06174=1038.286,203.644,-104.058,170.413,41.246,157.811
C06175=1038.281,203.395,-104.034,170.409,41.245,157.811
C06176=1038.275,203.147,-104.009,170.406,41.245,157.810
C06177=1038.269,202.898,-103.984,170.403,41.244,157.810
C06178=1038.263,202.649,-103.958,170.399,41.243,157.810
C06179=1038.257,202.400,-103.934,170.396,41.243,157.809
C06180=1038.250,202.151,-103.908,170.394,41.242,157.809
C06181=1038.244,201.903,-103.883,170.390,41.241,157.809
C06182=1038.238,201.654,-103.858,170.387,41.241,157.809
C06183=1038.233,201.405,-103.833,170.384,41.240,157.808
C06184=1038.226,201.157,-103.809,170.381,41.240,157.808
C06185=1038.220,200.908,-103.783,170.377,41.239,157.808
C06186=1038.214,200.659,-103.759,170.374,41.239,157.807
C06187=1038.207,200.410,-103.733,170.372,41.238,157.807
C06188=1038.201,200.162,-103.709,170.369,41.238,157.807
C06189=1038.195,199.913,-103.684,170.365,41.237,157.807
C06190=1038.188,199.665,-103.660,170.362,41.237,157.806
C06191=1038.182,199.416,-103.635,170.359,41.237,157.806
C06192=1038.175,199.167,-103.610,170.356,41.236,157.806
C06193=1038.170,198.918,-103.586,170.353,41.236,157.806
C06194=1038.163,198.670,-103.561,170.350,41.235,157.805
C06195=1038.157,198.421,-103.537,170.347,41.234,157.805
C06196=1038.151,198.173,-103.511,170.344,41.234,157.805
C06197=1038.144,197.924,-103.487,170.340,41.234,157.805
C06198=1038.138,197.675,-103.462,170.337,41.234,157.804
C06199=1038.132,197.426,-103.438,170.335,41.233,157.804
C06200=1038.126,197.178,-103.413,170.332,41.232,157.804
C06201=1038.119,196.929,-103.389,170.328,41.232,157.804
C06202=1038.113,196.680,-103.363,170.325,41.232,157.803
C06203=1038.107,196.431,-103.339,170.322,41.231,157.803
C06204=1038.101,196.183,-103.315,170.319,41.231,157.803
C06205=1038.095,195.934,-103.290,170.316,41.230,157.803
C06206=1038.088,195.685,-103.266,170.313,41.230,157.802
C06207=1038.082,195.436,-103.240,170.310,41.229,157.802
C06208=1038.076,195.188,-103.217,170.307,41.229,157.802
C06209=1038.070,194.939,-103.192,170.304,41.229,157.802
C06210=1038.063,194.690,-103.167,170.301,41.228,157.801
C06211=1038.058,194.442,-103.143,170.298,41.227,157.801
C06212=1038.051,194.193,-103.119,170.295,41.227,157.801
C06213=1038.045,193.944,-103.094,170.292,41.227,157.801
C06214=1038.039,193.696,-103.070,170.289,41.227,157.800
C06215=1038.033,193.447,-103.046,170.286,41.226,157.800
C06216=1038.026,193.198,-103.021,170.283,41.225,157.800
C06217=1038.021,192.950,-102.997,170.280,41.225,157.800
C06218=1038.014,192.701,-102.973,170.277,41.225,157.799
C06219=1038.008,192.451,-102.948,170.274,41.225,157.799
C06220=1038.002,192.204,-102.924,170.271,41.224,157.799
C06221=1037.996,191.955,-102.899,170.268,41.223,157.799
C06222=1037.990,191.706,-102.875,170.265,41.223,157.798
C06223=1037.984,191.457,-102.851,170.262,41.223,157.798
C06224=1037.978,191.208,-102.826,170.259,41.223,157.798
C06225=1037.972,190.960,-102.802,170.256,41.222,157.798
C06226=1037.966,190.711,-102.777,170.253,41.221,157.797
C06227=1037.959,190.462,-102.753,170.250,41.221,157.797
C06228=1037.954,190.213,-102.729,170.247,41.221,157.797
C06229=1037.948,189.964,-102.705,170.245,41.220,157.797
C06230=1037.942,189.716,-102.680,170.242,41.220,157.796
C06231=1037.932,189.299,-102.640,170.236,41.219,157.796
C06232=1037.921,188.883,-102.599,170.232,41.219,157.796
C06233=1037.911,188.467,-102.559,170.226,41.218,157.795
C06234=1037.901,188.050,-102.518,170.222,41.217,157.795
C06235=1037.895,187.801,-102.493,170.219,41.217,157.795
C06236=1037.889,187.552,-102.469,170.216,41.217,157.794
C06237=1037.884,187.304,-102.445,170.213,41.216,157.794
C06238=1037.877,187.055,-102.421,170.210,41.216,157.794
C06239=1037.872,186.806,-102.397,170.207,41.215,157.794
C06240=1037.865,186.557,-102.373,170.205,41.215,157.793
C06241=1037.859,186.309,-102.349,170.202,41.215,157.793
C06242=1037.853,186.060,-102.325,170.198,41.214,157.793
C06243=1037.847,185.811,-102.301,170.196,41.214,157.793
C06244=1037.841,185.562,-102.276,170.193,41.214,157.793
C06245=1037.835,185.314,-102.253,170.190,41.213,157.792
C06246=1037.830,185.065,-102.228,170.187,41.212,157.792
C06247=1037.823,184.816,-102.204,170.184,41.212,157.792
C06248=1037.818,184.568,-102.180,170.182,41.212,157.792
C06249=1037.811,184.319,-102.156,170.179,41.212,157.791
C06250=1037.806,184.070,-102.133,170.176,41.211,157.791
C06251=1037.800,183.821,-102.109,170.173,41.211,157.791
C06252=1037.794,183.572,-102.084,170.170,41.211,157.791
C06253=1037.788,183.323,-102.060,170.167,41.210,157.790
C06254=1037.782,183.075,-102.037,170.165,41.210,157.790
C06255=1037.775,182.825,-102.013,170.162,41.210,157.790
C06256=1037.769,182.577,-101.990,170.158,41.210,157.790
C06257=1037.763,182.328,-101.966,170.156,41.209,157.790
C06258=1037.756,182.079,-101.943,170.153,41.210,157.790
C06259=1037.749,181.830,-101.919,170.150,41.209,157.789
C06260=1037.743,181.582,-101.896,170.148,41.209,157.789
C06261=1037.737,181.332,-101.872,170.145,41.209,157.789
C06262=1037.731,181.084,-101.849,170.142,41.209,157.789
C06263=1037.724,180.835,-101.825,170.138,41.209,157.789
C06264=1037.719,180.586,-101.802,170.136,41.208,157.788
C06265=1037.712,180.337,-101.778,170.133,41.208,157.788
C06266=1037.706,180.088,-101.755,170.130,41.208,157.788
C06267=1037.700,179.839,-101.731,170.128,41.208,157.788
C06268=1037.693,179.591,-101.708,170.125,41.208,157.788
C06269=1037.687,179.343,-101.685,170.121,41.208,157.787
C06270=1037.680,179.094,-101.661,170.119,41.207,157.787
C06271=1037.675,178.845,-101.638,170.116,41.208,157.787
C06272=1037.668,178.596,-101.614,170.113,41.207,157.787
C06273=1037.662,178.347,-101.591,170.111,41.207,157.787
C06274=1037.656,178.098,-101.567,170.107,41.207,157.786
C06275=1037.650,177.849,-101.544,170.105,41.206,157.786
C06276=1037.643,177.601,-101.521,170.102,41.207,157.786
C06277=1037.637,177.351,-101.497,170.099,41.206,157.786
C06278=1037.631,177.103,-101.474,170.097,41.206,157.786
C06279=1037.622,176.738,-101.439,170.093,41.206,157.786
C06280=1037.613,176.372,-101.405,170.088,41.206,157.785
C06281=1037.604,176.007,-101.371,170.084,41.206,157.785
C06282=1037.595,175.642,-101.337,170.080,41.205,157.785
C06283=1037.588,175.392,-101.314,170.078,41.205,157.785
C06284=1037.582,175.144,-101.290,170.075,41.205,157.784
C06285=1037.577,174.895,-101.267,170.072,41.205,157.784
C06286=1037.570,174.645,-101.244,170.069,41.205,157.784
C06287=1037.564,174.397,-101.220,170.066,41.205,157.784
C06288=1037.558,174.148,-101.198,170.064,41.204,157.784
C06289=1037.551,173.900,-101.174,170.061,41.205,157.784
C06290=1037.545,173.651,-101.151,170.059,41.204,157.783
C06291=1037.539,173.366,-101.124,170.056,41.204,157.783
C06292=1037.531,173.081,-101.098,170.052,41.204,157.783
C06293=1037.525,172.797,-101.071,170.049,41.203,157.783
C06294=1037.517,172.512,-101.045,170.046,41.204,157.783
C06295=1037.512,172.263,-101.022,170.043,41.204,157.782
C06296=1037.506,172.015,-100.998,170.041,41.203,157.782
C06297=1037.499,171.766,-100.975,170.038,41.203,157.782
C06298=1037.493,171.517,-100.952,170.035,41.203,157.782
C06299=1037.487,171.268,-100.929,170.032,41.203,157.782
C06300=1037.481,171.019,-100.906,170.029,41.203,157.781
C06301=1037.475,170.770,-100.882,170.027,41.203,157.781
C06302=1037.469,170.521,-100.859,170.024,41.203,157.781
C06303=1037.463,170.272,-100.837,170.022,41.202,157.781
C06304=1037.457,170.023,-100.814,170.019,41.203,157.781
C06305=1037.450,169.775,-100.790,170.016,41.202,157.781
C06306=1037.445,169.526,-100.767,170.013,41.202,157.780
C06307=1037.439,169.277,-100.744,170.011,41.202,157.780
C06308=1037.433,169.028,-100.721,170.008,41.202,157.780
C06309=1037.427,168.779,-100.699,170.006,41.202,157.780
C06310=1037.421,168.531,-100.675,170.003,41.201,157.780
C06311=1037.414,168.281,-100.652,170.001,41.202,157.780
C06312=1037.408,168.032,-100.629,169.997,41.201,157.779
C06313=1037.403,167.784,-100.606,169.994,41.201,157.779
C06314=1037.396,167.535,-100.584,169.992,41.201,157.779
C06315=1037.391,167.286,-100.561,169.989,41.201,157.779
C06316=1037.385,167.037,-100.538,169.987,41.201,157.779
C06317=1037.378,166.788,-100.514,169.984,41.200,157.779
C06318=1037.373,166.539,-100.492,169.982,41.201,157.778
C06319=1037.366,166.291,-100.468,169.978,41.200,157.778
C06320=1037.360,166.042,-100.446,169.976,41.200,157.778
C06321=1037.355,165.793,-100.423,169.973,41.200,157.778
C06322=1037.349,165.544,-100.400,169.971,41.200,157.778
C06323=1037.343,165.295,-100.377,169.969,41.200,157.778
C06324=1037.337,165.047,-100.354,169.966,41.200,157.778
C06325=1037.331,164.798,-100.331,169.964,41.200,157.777
C06326=1037.325,164.549,-100.308,169.960,41.199,157.777
C06327=1037.319,164.299,-100.285,169.958,41.199,157.777
C06328=1037.313,164.050,-100.262,169.955,41.199,157.777
C06329=1037.307,163.802,-100.240,169.953,41.199,157.777
C06330=1037.301,163.553,-100.217,169.950,41.199,157.777
C06331=1037.295,163.304,-100.194,169.948,41.199,157.776
C06332=1037.289,163.055,-100.171,169.945,41.199,157.776
C06333=1037.283,162.806,-100.149,169.942,41.198,157.776
C06334=1037.277,162.558,-100.126,169.939,41.199,157.776
C06335=1037.272,162.308,-100.103,169.937,41.198,157.776
C06336=1037.266,162.059,-100.081,169.935,41.198,157.775
C06337=1037.260,161.810,-100.058,169.932,41.198,157.775
C06338=1037.254,161.562,-100.035,169.930,41.198,157.775
C06339=1037.248,161.313,-100.012,169.926,41.197,157.775
C06340=1037.242,161.064,-99.989,169.924,41.198,157.775
C06341=1037.237,160.815,-99.966,169.921,41.197,157.775
C06342=1037.230,160.566,-99.944,169.919,41.197,157.774
C06343=1037.224,160.317,-99.921,169.917,41.197,157.774
C06344=1037.219,160.068,-99.899,169.914,41.197,157.774
C06345=1037.213,159.819,-99.877,169.912,41.197,157.774
C06346=1037.207,159.570,-99.854,169.909,41.197,157.774
C06347=1037.200,159.322,-99.831,169.907,41.197,157.774
C06348=1037.194,159.073,-99.810,169.903,41.197,157.774
C06349=1037.188,158.824,-99.787,169.901,41.197,157.774
C06350=1037.182,158.575,-99.764,169.898,41.197,157.773
C06351=1037.177,158.326,-99.742,169.896,41.197,157.773
C06352=1037.170,158.077,-99.720,169.893,41.197,157.773
C06353=1037.164,157.828,-99.697,169.891,41.197,157.773
C06354=1037.158,157.579,-99.675,169.888,41.198,157.773
C06355=1037.151,157.294,-99.649,169.886,41.197,157.773
C06356=1037.144,157.009,-99.624,169.883,41.197,157.772
C06357=1037.137,156.724,-99.598,169.879,41.197,157.772
C06358=1037.130,156.438,-99.573,169.876,41.197,157.772
C06359=1037.124,156.190,-99.551,169.874,41.197,157.772
C06360=1037.117,155.941,-99.528,169.871,41.198,157.772
C06361=1037.112,155.692,-99.506,169.869,41.197,157.772
C06362=1037.105,155.443,-99.484,169.866,41.198,157.772
C06363=1037.099,155.194,-99.462,169.864,41.197,157.772
C06364=1037.093,154.945,-99.439,169.862,41.198,157.771
C06365=1037.087,154.696,-99.418,169.859,41.197,157.771
C06366=1037.081,154.447,-99.395,169.857,41.198,157.771
C06367=1037.075,154.198,-99.373,169.854,41.198,157.771
C06368=1037.069,153.949,-99.351,169.851,41.198,157.771
C06369=1037.063,153.700,-99.329,169.848,41.198,157.771
C06370=1037.056,153.451,-99.307,169.846,41.198,157.771
C06371=1037.051,153.202,-99.284,169.844,41.198,157.771
C06372=1037.044,152.953,-99.262,169.841,41.198,157.770
C06373=1037.038,152.704,-99.240,169.839,41.198,157.770
C06374=1037.032,152.456,-99.218,169.836,41.198,157.770
C06375=1037.026,152.206,-99.196,169.834,41.198,157.770
C06376=1037.020,151.957,-99.174,169.831,41.198,157.770
C06377=1037.014,151.708,-99.152,169.829,41.198,157.770
C06378=1037.008,151.460,-99.131,169.826,41.198,157.770
C06379=1037.002,151.211,-99.108,169.823,41.198,157.770
C06380=1036.995,150.962,-99.087,169.821,41.199,157.769
C06381=1036.990,150.712,-99.064,169.818,41.198,157.769
C06382=1036.984,150.464,-99.042,169.816,41.199,157.769
C06383=1036.977,150.215,-99.020,169.814,41.199,157.769
C06384=1036.971,149.966,-98.998,169.811,41.199,157.769
C06385=1036.965,149.717,-98.976,169.809,41.199,157.769
C06386=1036.959,149.468,-98.955,169.806,41.199,157.769
C06387=1036.953,149.219,-98.932,169.804,41.199,157.769
C06388=1036.947,148.970,-98.911,169.802,41.199,157.769
C06389=1036.941,148.721,-98.889,169.798,41.199,157.768
C06390=1036.935,148.472,-98.867,169.796,41.199,157.768
C06391=1036.928,148.223,-98.845,169.794,41.199,157.768
C06392=1036.922,147.974,-98.823,169.791,41.199,157.768
C06393=1036.916,147.725,-98.802,169.789,41.199,157.768
C06394=1036.911,147.476,-98.780,169.786,41.200,157.768
C06395=1036.904,147.228,-98.758,169.784,41.200,157.768
C06396=1036.898,146.979,-98.736,169.782,41.199,157.768
C06397=1036.893,146.729,-98.714,169.779,41.200,157.767
C06398=1036.886,146.480,-98.693,169.777,41.200,157.767
C06399=1036.879,146.231,-98.672,169.774,41.200,157.767
C06400=1036.873,145.982,-98.649,169.772,41.200,157.767
C06401=1036.867,145.734,-98.628,169.770,41.200,157.767
C06402=1036.861,145.485,-98.606,169.767,41.201,157.767
C06403=1036.855,145.235,-98.585,169.764,41.200,157.767
C06404=1036.849,144.986,-98.563,169.761,41.201,157.767
C06405=1036.843,144.737,-98.541,169.759,41.201,157.767
C06406=1036.837,144.488,-98.520,169.757,41.201,157.767
C06407=1036.831,144.239,-98.498,169.754,41.201,157.766
C06408=1036.825,143.991,-98.476,169.752,41.201,157.766
C06409=1036.818,143.741,-98.454,169.750,41.201,157.766
C06410=1036.812,143.492,-98.433,169.747,41.202,157.766
C06411=1036.805,143.243,-98.412,169.745,41.202,157.766
C06412=1036.800,142.995,-98.391,169.742,41.202,157.766
C06413=1036.794,142.746,-98.369,169.740,41.202,157.766
C06414=1036.787,142.496,-98.347,169.738,41.202,157.766
C06415=1036.781,142.247,-98.326,169.735,41.203,157.766
C06416=1036.776,141.999,-98.304,169.732,41.202,157.765
C06417=1036.770,141.750,-98.283,169.730,41.202,157.765
C06418=1036.763,141.500,-98.261,169.727,41.203,157.765
C06419=1036.756,141.216,-98.237,169.725,41.203,157.765
C06420=1036.749,140.929,-98.212,169.722,41.203,157.765
C06421=1036.743,140.644,-98.187,169.719,41.203,157.765
C06422=1036.736,140.359,-98.163,169.717,41.203,157.765
C06423=1036.730,140.109,-98.142,169.714,41.203,157.765
C06424=1036.723,139.860,-98.120,169.712,41.203,157.765
C06425=1036.717,139.611,-98.099,169.710,41.204,157.764
C06426=1036.712,139.363,-98.077,169.707,41.204,157.764
C06427=1036.705,139.113,-98.056,169.705,41.204,157.764
C06428=1036.699,138.864,-98.035,169.703,41.204,157.764
C06429=1036.692,138.615,-98.013,169.700,41.204,157.764
C06430=1036.687,138.367,-97.992,169.698,41.205,157.764
C06431=1036.681,138.118,-97.970,169.696,41.205,157.764
C06432=1036.674,137.868,-97.950,169.693,41.205,157.764
C06433=1036.669,137.620,-97.928,169.690,41.205,157.764
C06434=1036.662,137.370,-97.907,169.688,41.205,157.764
C06435=1036.656,137.121,-97.885,169.685,41.205,157.764
C06436=1036.650,136.873,-97.865,169.683,41.206,157.763
C06437=1036.644,136.624,-97.843,169.681,41.206,157.763
C06438=1036.638,136.374,-97.822,169.678,41.206,157.763
C06439=1036.631,136.125,-97.801,169.676,41.206,157.763
C06440=1036.625,135.877,-97.780,169.674,41.206,157.763
C06441=1036.619,135.627,-97.758,169.671,41.206,157.763
C06442=1036.613,135.378,-97.738,169.669,41.207,157.763
C06443=1036.607,135.129,-97.716,169.667,41.207,157.763
C06444=1036.601,134.880,-97.695,169.664,41.207,157.763
C06445=1036.594,134.631,-97.674,169.662,41.208,157.763
C06446=1036.589,134.382,-97.653,169.660,41.208,157.763
C06447=1036.583,134.133,-97.632,169.657,41.208,157.762
C06448=1036.576,133.884,-97.611,169.655,41.208,157.762
C06449=1036.570,133.635,-97.590,169.653,41.208,157.762
C06450=1036.564,133.386,-97.569,169.650,41.208,157.762
C06451=1036.557,133.137,-97.547,169.647,41.209,157.762
C06452=1036.552,132.888,-97.527,169.645,41.209,157.762
C06453=1036.545,132.639,-97.506,169.642,41.209,157.762
C06454=1036.540,132.390,-97.484,169.640,41.209,157.762
C06455=1036.534,132.140,-97.464,169.638,41.209,157.762
C06456=1036.527,131.891,-97.442,169.636,41.209,157.762
C06457=1036.521,131.643,-97.421,169.633,41.210,157.762
C06458=1036.515,131.393,-97.400,169.631,41.210,157.762
C06459=1036.509,131.145,-97.380,169.629,41.210,157.761
C06460=1036.503,130.895,-97.359,169.626,41.211,157.761
C06461=1036.496,130.646,-97.338,169.624,41.211,157.761
C06462=1036.490,130.397,-97.318,169.622,41.211,157.761
C06463=1036.484,130.148,-97.296,169.619,41.212,157.761
C06464=1036.478,129.899,-97.276,169.617,41.212,157.761
C06465=1036.471,129.651,-97.255,169.615,41.212,157.761
C06466=1036.466,129.401,-97.234,169.612,41.212,157.761
C06467=1036.459,129.153,-97.213,169.610,41.213,157.761
C06468=1036.453,128.903,-97.193,169.608,41.213,157.761
C06469=1036.446,128.654,-97.172,169.605,41.213,157.761
C06470=1036.440,128.405,-97.152,169.603,41.213,157.761
C06471=1036.434,128.156,-97.131,169.601,41.214,157.761
C06472=1036.428,127.906,-97.110,169.599,41.214,157.761
C06473=1036.422,127.657,-97.090,169.596,41.214,157.760
C06474=1036.415,127.409,-97.069,169.594,41.215,157.760
C06475=1036.410,127.159,-97.048,169.592,41.215,157.760
C06476=1036.403,126.911,-97.027,169.589,41.215,157.760
C06477=1036.397,126.662,-97.007,169.587,41.215,157.760
C06478=1036.391,126.412,-96.986,169.585,41.216,157.760
C06479=1036.384,126.163,-96.965,169.582,41.216,157.760
C06480=1036.378,125.914,-96.945,169.580,41.216,157.760
C06481=1036.372,125.665,-96.923,169.578,41.217,157.760
C06482=1036.366,125.416,-96.904,169.575,41.217,157.760
C06483=1036.359,125.131,-96.880,169.572,41.217,157.760
C06484=1036.351,124.845,-96.856,169.569,41.218,157.760
C06485=1036.344,124.559,-96.833,169.567,41.218,157.760
C06486=1036.337,124.273,-96.809,169.564,41.218,157.760
C06487=1036.331,124.024,-96.789,169.562,41.218,157.759
C06488=1036.325,123.776,-96.768,169.559,41.219,157.759
C06489=1036.319,123.526,-96.747,169.557,41.219,157.759
C06490=1036.313,123.277,-96.727,169.555,41.219,157.759
C06491=1036.306,123.028,-96.706,169.553,41.220,157.759
C06492=1036.300,122.779,-96.686,169.550,41.220,157.759
C06493=1036.294,122.529,-96.665,169.548,41.220,157.759
C06494=1036.288,122.281,-96.646,169.546,41.220,157.759
C06495=1036.281,122.032,-96.624,169.544,41.221,157.759
C06496=1036.276,121.783,-96.604,169.541,41.221,157.759
C06497=1036.270,121.534,-96.584,169.539,41.221,157.759
C06498=1036.263,121.284,-96.564,169.537,41.222,157.759
C06499=1036.257,121.036,-96.543,169.535,41.222,157.759
C06500=1036.251,120.786,-96.522,169.532,41.222,157.759
C06501=1036.245,120.537,-96.502,169.530,41.222,157.758
C06502=1036.238,120.288,-96.482,169.528,41.222,157.758
C06503=1036.232,120.039,-96.462,169.526,41.222,157.758
C06504=1036.226,119.790,-96.440,169.523,41.223,157.758
C06505=1036.220,119.541,-96.420,169.521,41.223,157.758
C06506=1036.214,119.292,-96.400,169.519,41.223,157.758
C06507=1036.208,119.042,-96.379,169.517,41.223,157.758
C06508=1036.202,118.794,-96.359,169.514,41.224,157.758
C06509=1036.196,118.544,-96.339,169.512,41.224,157.758
C06510=1036.190,118.295,-96.319,169.510,41.224,157.758
C06511=1036.184,118.047,-96.298,169.508,41.225,157.758
C06512=1036.178,117.797,-96.277,169.504,41.225,157.758
C06513=1036.172,117.548,-96.258,169.502,41.225,157.758
C06514=1036.165,117.299,-96.237,169.500,41.225,157.757
C06515=1036.160,117.050,-96.217,169.498,41.226,157.757
C06516=1036.154,116.801,-96.197,169.496,41.226,157.757
C06517=1036.147,116.551,-96.176,169.493,41.226,157.757
C06518=1036.141,116.303,-96.156,169.491,41.227,157.757
C06519=1036.136,116.054,-96.136,169.489,41.227,157.757
C06520=1036.129,115.804,-96.116,169.487,41.227,157.757
C06521=1036.123,115.555,-96.096,169.484,41.227,157.757
C06522=1036.117,115.306,-96.075,169.482,41.228,157.757
C06523=1036.111,115.057,-96.054,169.480,41.228,157.757
C06524=1036.105,114.808,-96.034,169.478,41.228,157.757
C06525=1036.099,114.559,-96.014,169.476,41.228,157.757
C06526=1036.093,114.310,-95.994,169.473,41.228,157.756
C06527=1036.087,114.061,-95.973,169.471,41.228,157.756
C06528=1036.081,113.811,-95.953,169.469,41.229,157.756
C06529=1036.075,113.563,-95.933,169.467,41.229,157.756
C06530=1036.069,113.314,-95.913,169.465,41.229,157.756
C06531=1036.063,113.064,-95.894,169.462,41.229,157.756
C06532=1036.057,112.815,-95.873,169.460,41.230,157.756
C06533=1036.051,112.566,-95.853,169.458,41.230,157.756
C06534=1036.044,112.316,-95.833,169.456,41.230,157.756
C06535=1036.038,112.068,-95.813,169.453,41.231,157.756
C06536=1036.032,111.819,-95.793,169.451,41.231,157.756
C06537=1036.025,111.569,-95.773,169.449,41.232,157.756
C06538=1036.019,111.321,-95.753,169.447,41.232,157.756
C06539=1036.014,111.071,-95.734,169.445,41.232,157.756
C06540=1036.007,110.822,-95.713,169.442,41.233,157.756
C06541=1036.001,110.573,-95.693,169.440,41.233,157.756
C06542=1035.995,110.324,-95.673,169.438,41.233,157.756
C06543=1035.989,110.074,-95.653,169.436,41.233,157.755
C06544=1035.983,109.825,-95.634,169.433,41.234,157.755
C06545=1035.977,109.576,-95.614,169.431,41.234,157.755
C06546=1035.970,109.327,-95.594,169.429,41.235,157.755
C06547=1035.963,109.041,-95.571,169.426,41.235,157.755
C06548=1035.955,108.755,-95.549,169.424,41.235,157.755
C06549=1035.949,108.469,-95.526,169.421,41.236,157.755
C06550=1035.941,108.184,-95.504,169.419,41.236,157.755
C06551=1035.935,107.935,-95.484,169.416,41.236,157.755
C06552=1035.929,107.686,-95.464,169.414,41.237,157.755
C06553=1035.922,107.436,-95.445,169.412,41.238,157.755
C06554=1035.916,107.187,-95.425,169.410,41.238,157.755
C06555=1035.910,106.938,-95.405,169.407,41.238,157.755
C06556=1035.905,106.689,-95.385,169.405,41.238,157.755
C06557=1035.898,106.440,-95.365,169.403,41.239,157.755
C06558=1035.891,106.191,-95.346,169.401,41.239,157.755
C06559=1035.886,105.942,-95.327,169.399,41.239,157.755
C06560=1035.880,105.693,-95.307,169.395,41.240,157.755
C06561=1035.873,105.443,-95.286,169.394,41.241,157.755
C06562=1035.867,105.194,-95.267,169.392,41.241,157.755
C06563=1035.861,104.945,-95.248,169.390,41.241,157.754
C06564=1035.855,104.697,-95.228,169.388,41.241,157.754
C06565=1035.848,104.446,-95.208,169.385,41.242,157.754
C06566=1035.842,104.198,-95.188,169.382,41.242,157.754
C06567=1035.837,103.948,-95.169,169.380,41.242,157.754
C06568=1035.830,103.700,-95.150,169.378,41.242,157.754
C06569=1035.824,103.450,-95.130,169.375,41.243,157.754
C06570=1035.818,103.201,-95.110,169.374,41.244,157.754
C06571=1035.812,102.952,-95.090,169.372,41.244,157.754
C06572=1035.806,102.702,-95.071,169.369,41.244,157.754
C06573=1035.799,102.454,-95.051,169.367,41.244,157.754
C06574=1035.793,102.205,-95.032,169.365,41.245,157.754
C06575=1035.787,101.955,-95.012,169.362,41.245,157.754
C06576=1035.781,101.706,-94.993,169.360,41.245,157.754
C06577=1035.774,101.457,-94.973,169.358,41.245,157.754
C06578=1035.769,101.208,-94.954,169.356,41.246,157.754
C06579=1035.763,100.959,-94.934,169.354,41.246,157.754
C06580=1035.757,100.709,-94.915,169.351,41.246,157.753
C06581=1035.750,100.460,-94.895,169.349,41.247,157.753
C06582=1035.744,100.211,-94.876,169.347,41.248,157.753
C06583=1035.738,99.962,-94.856,169.345,41.248,157.753
C06584=1035.732,99.713,-94.837,169.343,41.248,157.753
C06585=1035.726,99.464,-94.817,169.340,41.248,157.753
C06586=1035.719,99.215,-94.799,169.338,41.249,157.753
C06587=1035.713,98.965,-94.779,169.336,41.250,157.753
C06588=1035.706,98.716,-94.760,169.334,41.250,157.753
C06589=1035.700,98.467,-94.740,169.331,41.250,157.753
C06590=1035.694,98.218,-94.722,169.329,41.250,157.753
C06591=1035.688,97.969,-94.702,169.327,41.251,157.753
C06592=1035.681,97.719,-94.683,169.325,41.252,157.753
C06593=1035.675,97.470,-94.663,169.323,41.252,157.753
C06594=1035.669,97.221,-94.644,169.320,41.252,157.753
C06595=1035.663,96.972,-94.625,169.318,41.252,157.753
C06596=1035.657,96.723,-94.606,169.316,41.253,157.753
C06597=1035.651,96.474,-94.586,169.314,41.254,157.753
C06598=1035.644,96.225,-94.568,169.312,41.254,157.753
C06599=1035.638,95.975,-94.548,169.309,41.254,157.753
C06600=1035.631,95.726,-94.529,169.307,41.254,157.753
C06601=1035.625,95.477,-94.509,169.306,41.255,157.753
C06602=1035.619,95.227,-94.491,169.303,41.256,157.753
C06603=1035.613,94.978,-94.472,169.301,41.256,157.753
C06604=1035.607,94.730,-94.452,169.298,41.256,157.752
C06605=1035.601,94.480,-94.433,169.296,41.256,157.752
C06606=1035.594,94.231,-94.414,169.295,41.257,157.752
C06607=1035.589,93.982,-94.395,169.293,41.258,157.752
C06608=1035.582,93.733,-94.376,169.291,41.258,157.752
C06609=1035.576,93.484,-94.356,169.287,41.258,157.752
C06610=1035.569,93.234,-94.337,169.285,41.258,157.752
C06611=1035.562,92.949,-94.315,169.283,41.259,157.752
C06612=1035.555,92.662,-94.294,169.281,41.260,157.752
C06613=1035.548,92.377,-94.271,169.279,41.260,157.752
C06614=1035.541,92.091,-94.250,169.275,41.260,157.752
C06615=1035.536,91.842,-94.231,169.273,41.261,157.752
C06616=1035.529,91.593,-94.212,169.271,41.261,157.752
C06617=1035.524,91.343,-94.193,169.269,41.261,157.752
C06618=1035.517,91.095,-94.174,169.268,41.262,157.752
C06619=1035.511,90.845,-94.154,169.265,41.262,157.752
C06620=1035.504,90.595,-94.135,169.262,41.263,157.752
C06621=1035.498,90.346,-94.116,169.260,41.263,157.752
C06622=1035.492,90.097,-94.098,169.258,41.263,157.752
C06623=1035.486,89.847,-94.078,169.256,41.263,157.752
C06624=1035.480,89.598,-94.060,169.254,41.264,157.752
C06625=1035.473,89.349,-94.041,169.252,41.265,157.751
C06626=1035.467,89.100,-94.022,169.249,41.265,157.751
C06627=1035.461,88.851,-94.004,169.248,41.266,157.752
C06628=1035.455,88.601,-93.984,169.246,41.266,157.751
C06629=1035.448,88.352,-93.966,169.243,41.266,157.751
C06630=1035.442,88.103,-93.947,169.241,41.267,157.751
C06631=1035.436,87.854,-93.928,169.239,41.268,157.751
C06632=1035.429,87.605,-93.910,169.237,41.268,157.751
C06633=1035.423,87.356,-93.891,169.234,41.268,157.751
C06634=1035.417,87.106,-93.872,169.232,41.269,157.751
C06635=1035.411,86.857,-93.853,169.230,41.269,157.751
C06636=1035.404,86.608,-93.835,169.228,41.270,157.751
C06637=1035.398,86.359,-93.816,169.226,41.270,157.751
C06638=1035.391,86.110,-93.797,169.223,41.271,157.751
C06639=1035.386,85.861,-93.778,169.221,41.271,157.751
C06640=1035.379,85.611,-93.759,169.219,41.271,157.751
C06641=1035.373,85.362,-93.741,169.217,41.272,157.751
C06642=1035.366,85.113,-93.722,169.215,41.272,157.751
C06643=1035.360,84.864,-93.704,169.212,41.273,157.751
C06644=1035.354,84.614,-93.686,169.210,41.273,157.751
C06645=1035.348,84.365,-93.666,169.208,41.274,157.751
C06646=1035.342,84.116,-93.648,169.206,41.274,157.751
C06647=1035.335,83.867,-93.629,169.204,41.275,157.751
C06648=1035.329,83.617,-93.610,169.202,41.275,157.751
C06649=1035.322,83.368,-93.592,169.199,41.276,157.751
C06650=1035.317,83.119,-93.573,169.197,41.276,157.751
C06651=1035.311,82.869,-93.555,169.195,41.276,157.751
C06652=1035.304,82.620,-93.536,169.193,41.277,157.751
C06653=1035.298,82.371,-93.517,169.191,41.277,157.751
C06654=1035.292,82.123,-93.499,169.188,41.278,157.751
C06655=1035.286,81.873,-93.480,169.186,41.278,157.750
C06656=1035.279,81.624,-93.462,169.184,41.278,157.750
C06657=1035.274,81.374,-93.443,169.182,41.279,157.750
C06658=1035.267,81.125,-93.425,169.180,41.279,157.750
C06659=1035.261,80.876,-93.406,169.178,41.280,157.750
C06660=1035.254,80.627,-93.387,169.175,41.280,157.750
C06661=1035.248,80.378,-93.369,169.173,41.280,157.750
C06662=1035.242,80.128,-93.351,169.171,41.281,157.750
C06663=1035.236,79.879,-93.331,169.169,41.281,157.750
C06664=1035.230,79.630,-93.313,169.167,41.282,157.750
C06665=1035.224,79.381,-93.294,169.164,41.282,157.750
C06666=1035.218,79.131,-93.277,169.162,41.282,157.750
C06667=1035.211,78.882,-93.258,169.160,41.283,157.750
C06668=1035.205,78.633,-93.239,169.158,41.283,157.750
C06669=1035.199,78.383,-93.221,169.156,41.284,157.750
C06670=1035.193,78.134,-93.202,169.154,41.284,157.750
C06671=1035.187,77.885,-93.183,169.151,41.285,157.750
C06672=1035.181,77.636,-93.166,169.149,41.285,157.750
C06673=1035.175,77.387,-93.147,169.147,41.286,157.750
C06674=1035.168,77.137,-93.129,169.145,41.286,157.750
C06675=1035.161,76.851,-93.108,169.142,41.287,157.750
C06676=1035.154,76.566,-93.088,169.140,41.287,157.750
C06677=1035.146,76.279,-93.066,169.137,41.287,157.750
C06678=1035.139,75.994,-93.045,169.135,41.288,157.750
C06679=1035.133,75.745,-93.027,169.133,41.289,157.750
C06680=1035.127,75.495,-93.009,169.130,41.290,157.750
C06681=1035.120,75.246,-92.990,169.128,41.290,157.750
C06682=1035.115,74.997,-92.972,169.126,41.290,157.750
C06683=1035.108,74.748,-92.954,169.125,41.291,157.750
C06684=1035.101,74.498,-92.936,169.123,41.291,157.750
C06685=1035.095,74.249,-92.918,169.119,41.292,157.749
C06686=1035.089,73.999,-92.900,169.117,41.292,157.749
C06687=1035.082,73.750,-92.881,169.116,41.293,157.749
C06688=1035.077,73.501,-92.864,169.114,41.293,157.749
C06689=1035.070,73.252,-92.845,169.112,41.293,157.749
C06690=1035.064,73.002,-92.827,169.109,41.294,157.749
C06691=1035.058,72.753,-92.808,169.107,41.295,157.749
C06692=1035.051,72.504,-92.791,169.105,41.295,157.749
C06693=1035.045,72.255,-92.773,169.103,41.296,157.749
C06694=1035.039,72.006,-92.755,169.101,41.296,157.749
C06695=1035.033,71.757,-92.736,169.099,41.296,157.749
C06696=1035.027,71.507,-92.718,169.096,41.297,157.749
C06697=1035.020,71.258,-92.700,169.094,41.297,157.749
C06698=1035.015,71.009,-92.682,169.092,41.298,157.749
C06699=1035.008,70.759,-92.665,169.090,41.298,157.749
C06700=1035.001,70.510,-92.646,169.088,41.299,157.749
C06701=1034.995,70.260,-92.628,169.085,41.299,157.749
C06702=1034.989,70.012,-92.610,169.083,41.299,157.749
C06703=1034.983,69.762,-92.592,169.081,41.300,157.749
C06704=1034.977,69.512,-92.574,169.079,41.301,157.749
C06705=1034.970,69.264,-92.556,169.077,41.301,157.749
C06706=1034.964,69.014,-92.538,169.074,41.301,157.749
C06707=1034.958,68.766,-92.520,169.072,41.302,157.749
C06708=1034.952,68.516,-92.502,169.070,41.302,157.749
C06709=1034.945,68.266,-92.484,169.068,41.303,157.749
C06710=1034.939,68.017,-92.467,169.066,41.304,157.749
C06711=1034.933,67.768,-92.448,169.063,41.304,157.749
C06712=1034.926,67.519,-92.431,169.061,41.305,157.749
C06713=1034.920,67.269,-92.413,169.059,41.305,157.749
C06714=1034.914,67.020,-92.394,169.057,41.305,157.749
C06715=1034.907,66.771,-92.377,169.055,41.306,157.749
C06716=1034.901,66.521,-92.359,169.052,41.307,157.749
C06717=1034.895,66.272,-92.342,169.050,41.307,157.749
C06718=1034.889,66.024,-92.324,169.048,41.308,157.749
C06719=1034.883,65.774,-92.306,169.046,41.308,157.749
C06720=1034.876,65.524,-92.288,169.044,41.308,157.748
C06721=1034.870,65.275,-92.271,169.041,41.309,157.748
C06722=1034.864,65.026,-92.252,169.039,41.310,157.748
C06723=1034.858,64.776,-92.234,169.037,41.310,157.748
C06724=1034.851,64.527,-92.217,169.036,41.311,157.748
C06725=1034.845,64.278,-92.200,169.034,41.311,157.748
C06726=1034.838,64.029,-92.182,169.030,41.311,157.748
C06727=1034.832,63.779,-92.164,169.029,41.312,157.748
C06728=1034.826,63.530,-92.146,169.027,41.312,157.748
C06729=1034.820,63.281,-92.129,169.025,41.313,157.748
C06730=1034.813,63.032,-92.111,169.022,41.314,157.748
C06731=1034.807,62.782,-92.093,169.020,41.315,157.748
C06732=1034.800,62.533,-92.076,169.018,41.315,157.748
C06733=1034.794,62.284,-92.059,169.016,41.316,157.748
C06734=1034.787,62.034,-92.041,169.013,41.316,157.748
C06735=1034.781,61.784,-92.024,169.011,41.317,157.748
C06736=1034.775,61.535,-92.006,169.009,41.317,157.748
C06737=1034.768,61.286,-91.989,169.007,41.318,157.748
C06738=1034.761,61.037,-91.972,169.004,41.319,157.748
C06739=1034.754,60.751,-91.952,169.002,41.320,157.748
C06740=1034.747,60.465,-91.932,168.999,41.320,157.748
C06741=1034.740,60.178,-91.911,168.997,41.321,157.748
C06742=1034.732,59.892,-91.892,168.994,41.321,157.748
C06743=1034.726,59.643,-91.874,168.992,41.322,157.748
C06744=1034.720,59.394,-91.857,168.990,41.322,157.748
C06745=1034.713,59.145,-91.840,168.988,41.323,157.748
C06746=1034.707,58.895,-91.822,168.986,41.324,157.748
C06747=1034.700,58.646,-91.805,168.984,41.325,157.748
C06748=1034.694,58.397,-91.787,168.982,41.325,157.748
C06749=1034.688,58.147,-91.770,168.980,41.326,157.748
C06750=1034.681,57.898,-91.753,168.977,41.326,157.748
C06751=1034.674,57.649,-91.735,168.975,41.326,157.748
C06752=1034.669,57.400,-91.718,168.973,41.327,157.748
C06753=1034.662,57.150,-91.700,168.971,41.327,157.748
C06754=1034.655,56.901,-91.683,168.968,41.328,157.748
C06755=1034.650,56.652,-91.665,168.966,41.329,157.748
C06756=1034.643,56.402,-91.648,168.964,41.330,157.748
C06757=1034.637,56.154,-91.631,168.962,41.330,157.748
C06758=1034.631,55.903,-91.614,168.959,41.331,157.748
C06759=1034.624,55.654,-91.597,168.957,41.331,157.748
C06760=1034.618,55.405,-91.580,168.955,41.331,157.748
C06761=1034.611,55.155,-91.562,168.953,41.332,157.748
C06762=1034.605,54.907,-91.545,168.950,41.333,157.748
C06763=1034.598,54.657,-91.527,168.948,41.334,157.748
C06764=1034.592,54.407,-91.509,168.946,41.334,157.748
C06765=1034.586,54.158,-91.493,168.945,41.335,157.748
C06766=1034.579,53.909,-91.476,168.942,41.335,157.748
C06767=1034.574,53.660,-91.458,168.939,41.335,157.748
C06768=1034.567,53.410,-91.441,168.938,41.336,157.748
C06769=1034.561,53.162,-91.424,168.936,41.337,157.748
C06770=1034.555,52.912,-91.406,168.934,41.337,157.748
C06771=1034.549,52.662,-91.390,168.931,41.338,157.748
C06772=1034.542,52.413,-91.372,168.929,41.338,157.748
C06773=1034.536,52.164,-91.355,168.927,41.339,157.748
C06774=1034.529,51.915,-91.337,168.925,41.339,157.748
C06775=1034.524,51.665,-91.321,168.923,41.340,157.748
C06776=1034.517,51.416,-91.304,168.920,41.341,157.748
C06777=1034.511,51.167,-91.286,168.918,41.341,157.748
C06778=1034.504,50.917,-91.269,168.916,41.342,157.748
C06779=1034.498,50.668,-91.253,168.914,41.342,157.748
C06780=1034.492,50.418,-91.235,168.911,41.342,157.747
C06781=1034.486,50.169,-91.218,168.909,41.343,157.748
C06782=1034.479,49.920,-91.200,168.907,41.343,157.747
C06783=1034.474,49.670,-91.184,168.905,41.344,157.748
C06784=1034.467,49.421,-91.166,168.903,41.345,157.747
C06785=1034.461,49.172,-91.149,168.900,41.345,157.747
C06786=1034.454,48.922,-91.133,168.898,41.346,157.747
C06787=1034.449,48.673,-91.115,168.896,41.346,157.747
C06788=1034.442,48.424,-91.098,168.894,41.346,157.747
C06789=1034.436,48.174,-91.082,168.891,41.347,157.747
C06790=1034.430,47.925,-91.064,168.889,41.348,157.747
C06791=1034.424,47.676,-91.047,168.887,41.348,157.747
C06792=1034.418,47.427,-91.030,168.885,41.349,157.747
C06793=1034.411,47.177,-91.013,168.883,41.349,157.747
C06794=1034.405,46.928,-90.995,168.880,41.349,157.747
C06795=1034.399,46.678,-90.979,168.878,41.350,157.747
C06796=1034.392,46.429,-90.962,168.876,41.351,157.747
C06797=1034.387,46.180,-90.945,168.874,41.351,157.747
C06798=1034.380,45.930,-90.928,168.873,41.352,157.747
C06799=1034.374,45.681,-90.911,168.869,41.352,157.747
C06800=1034.368,45.431,-90.894,168.867,41.352,157.747
C06801=1034.362,45.182,-90.877,168.866,41.353,157.747
C06802=1034.356,44.933,-90.860,168.864,41.354,157.747
C06803=1034.348,44.646,-90.840,168.861,41.354,157.747
C06804=1034.341,44.360,-90.821,168.859,41.355,157.747
C06805=1034.334,44.074,-90.801,168.856,41.355,157.747
C06806=1034.327,43.788,-90.782,168.854,41.355,157.747
C06807=1034.321,43.538,-90.765,168.851,41.356,157.747
C06808=1034.315,43.289,-90.748,168.849,41.357,157.747
C06809=1034.309,43.039,-90.732,168.847,41.357,157.747
C06810=1034.303,42.790,-90.714,168.845,41.358,157.747
C06811=1034.297,42.540,-90.698,168.842,41.358,157.747
C06812=1034.290,42.291,-90.681,168.840,41.359,157.747
C06813=1034.284,42.042,-90.664,168.838,41.359,157.747
C06814=1034.278,41.793,-90.648,168.836,41.360,157.747
C06815=1034.271,41.543,-90.631,168.833,41.361,157.747
C06816=1034.265,41.294,-90.615,168.831,41.362,157.747
C06817=1034.259,41.045,-90.598,168.829,41.362,157.747
C06818=1034.252,40.795,-90.581,168.827,41.363,157.747
C06819=1034.246,40.546,-90.564,168.824,41.363,157.747
C06820=1034.240,40.297,-90.548,168.822,41.363,157.747
C06821=1034.233,40.047,-90.531,168.820,41.364,157.747
C06822=1034.227,39.798,-90.514,168.818,41.365,157.747
C06823=1034.221,39.548,-90.498,168.815,41.366,157.747
C06824=1034.215,39.298,-90.481,168.813,41.366,157.746
C06825=1034.208,39.050,-90.464,168.812,41.367,157.747
C06826=1034.202,38.800,-90.448,168.810,41.367,157.746
C06827=1034.196,38.550,-90.431,168.806,41.367,157.746
C06828=1034.190,38.302,-90.415,168.805,41.368,157.746
C06829=1034.184,38.052,-90.398,168.803,41.369,157.746
C06830=1034.177,37.802,-90.382,168.801,41.369,157.746
C06831=1034.171,37.554,-90.365,168.798,41.370,157.746
C06832=1034.165,37.304,-90.348,168.796,41.370,157.746
C06833=1034.158,37.054,-90.332,168.794,41.371,157.746
C06834=1034.152,36.805,-90.316,168.792,41.371,157.746
C06835=1034.146,36.556,-90.299,168.789,41.372,157.746
C06836=1034.139,36.306,-90.283,168.787,41.373,157.746
C06837=1034.133,36.057,-90.266,168.785,41.373,157.746
C06838=1034.126,35.808,-90.251,168.782,41.374,157.746
C06839=1034.120,35.558,-90.234,168.780,41.375,157.746
C06840=1034.114,35.308,-90.218,168.778,41.376,157.746
C06841=1034.108,35.060,-90.201,168.775,41.376,157.746
C06842=1034.100,34.810,-90.185,168.773,41.377,157.746
C06843=1034.094,34.561,-90.168,168.771,41.377,157.746
C06844=1034.088,34.311,-90.152,168.769,41.378,157.746
C06845=1034.082,34.062,-90.136,168.766,41.378,157.746
C06846=1034.075,33.812,-90.120,168.765,41.379,157.746
C06847=1034.069,33.563,-90.104,168.763,41.380,157.746
C06848=1034.063,33.314,-90.087,168.760,41.381,157.746
C06849=1034.057,33.065,-90.070,168.758,41.381,157.746
C06850=1034.050,32.815,-90.054,168.756,41.382,157.746
C06851=1034.044,32.566,-90.038,168.754,41.382,157.746
C06852=1034.038,32.316,-90.022,168.751,41.383,157.746
C06853=1034.032,32.067,-90.006,168.749,41.383,157.746
C06854=1034.025,31.817,-89.990,168.747,41.384,157.746
C06855=1034.019,31.568,-89.973,168.744,41.385,157.746
C06856=1034.013,31.319,-89.957,168.742,41.386,157.746
C06857=1034.007,31.069,-89.941,168.740,41.386,157.746
C06858=1033.999,30.820,-89.925,168.737,41.387,157.746
C06859=1033.993,30.570,-89.909,168.735,41.387,157.746
C06860=1033.987,30.321,-89.892,168.733,41.388,157.746
C06861=1033.982,30.071,-89.876,168.731,41.388,157.746
C06862=1033.975,29.822,-89.860,168.728,41.389,157.746
C06863=1033.968,29.572,-89.844,168.726,41.390,157.746
C06864=1033.962,29.323,-89.828,168.725,41.390,157.746
C06865=1033.956,29.074,-89.811,168.721,41.391,157.746
C06866=1033.950,28.825,-89.796,168.720,41.392,157.746
C06867=1033.942,28.538,-89.777,168.718,41.392,157.746
C06868=1033.936,28.252,-89.758,168.715,41.393,157.746
C06869=1033.929,27.965,-89.740,168.712,41.393,157.746
C06870=1033.921,27.679,-89.721,168.710,41.394,157.746
C06871=1033.914,27.430,-89.705,168.707,41.395,157.746
C06872=1033.909,27.180,-89.689,168.705,41.396,157.746
C06873=1033.901,26.931,-89.673,168.703,41.397,157.746
C06874=1033.895,26.681,-89.657,168.700,41.397,157.746
C06875=1033.889,26.432,-89.641,168.698,41.398,157.746
C06876=1033.883,26.182,-89.626,168.696,41.398,157.746
C06877=1033.877,25.933,-89.609,168.693,41.399,157.746
C06878=1033.870,25.684,-89.594,168.691,41.399,157.746
C06879=1033.864,25.434,-89.577,168.689,41.400,157.746
C06880=1033.857,25.185,-89.562,168.686,41.401,157.746
C06881=1033.851,24.935,-89.545,168.684,41.402,157.746
C06882=1033.845,24.686,-89.530,168.683,41.402,157.746
C06883=1033.839,24.436,-89.514,168.680,41.403,157.746
C06884=1033.832,24.187,-89.498,168.678,41.404,157.746
C06885=1033.826,23.938,-89.482,168.676,41.404,157.746
C06886=1033.819,23.688,-89.466,168.673,41.405,157.746
C06887=1033.813,23.438,-89.451,168.671,41.405,157.746
C06888=1033.807,23.189,-89.435,168.669,41.406,157.746
C06889=1033.801,22.940,-89.419,168.666,41.407,157.746
C06890=1033.794,22.691,-89.403,168.664,41.407,157.746
C06891=1033.788,22.441,-89.387,168.662,41.408,157.746
C06892=1033.782,22.192,-89.372,168.659,41.409,157.746
C06893=1033.775,21.943,-89.356,168.657,41.410,157.746
C06894=1033.769,21.694,-89.340,168.655,41.410,157.746
C06895=1033.763,21.444,-89.325,168.652,41.411,157.746
C06896=1033.756,21.194,-89.308,168.650,41.411,157.746
C06897=1033.749,20.945,-89.293,168.648,41.412,157.746
C06898=1033.744,20.695,-89.277,168.645,41.413,157.746
C06899=1033.737,20.446,-89.261,168.644,41.413,157.746
C06900=1033.731,20.196,-89.245,168.642,41.414,157.746
C06901=1033.725,19.947,-89.230,168.639,41.415,157.746
C06902=1033.719,19.697,-89.214,168.637,41.416,157.746
C06903=1033.712,19.448,-89.198,168.635,41.416,157.746
C06904=1033.706,19.199,-89.183,168.632,41.417,157.746
C06905=1033.700,18.949,-89.167,168.630,41.417,157.746
C06906=1033.693,18.700,-89.152,168.628,41.418,157.746
C06907=1033.687,18.450,-89.136,168.625,41.419,157.746
C06908=1033.681,18.201,-89.120,168.623,41.419,157.746
C06909=1033.674,17.952,-89.105,168.620,41.420,157.746
C06910=1033.668,17.702,-89.089,168.618,41.421,157.746
C06911=1033.662,17.453,-89.074,168.616,41.422,157.746
C06912=1033.655,17.204,-89.058,168.613,41.423,157.746
C06913=1033.650,16.954,-89.043,168.611,41.423,157.746
C06914=1033.643,16.705,-89.027,168.610,41.424,157.746
C06915=1033.636,16.455,-89.012,168.607,41.424,157.746
C06916=1033.631,16.206,-88.996,168.605,41.425,157.746
C06917=1033.624,15.957,-88.980,168.603,41.425,157.746
C06918=1033.617,15.707,-88.965,168.600,41.426,157.746
C06919=1033.611,15.458,-88.950,168.598,41.427,157.746
C06920=1033.605,15.208,-88.934,168.595,41.428,157.746
C06921=1033.599,14.958,-88.919,168.593,41.429,157.746
C06922=1033.592,14.709,-88.904,168.591,41.429,157.746
C06923=1033.586,14.459,-88.888,168.588,41.430,157.746
C06924=1033.580,14.210,-88.872,168.586,41.430,157.746
C06925=1033.573,13.961,-88.857,168.584,41.431,157.746
C06926=1033.567,13.711,-88.841,168.581,41.432,157.746
C06927=1033.561,13.462,-88.826,168.579,41.432,157.746
C06928=1033.555,13.212,-88.811,168.576,41.433,157.746
C06929=1033.548,12.963,-88.796,168.575,41.434,157.746
C06930=1033.542,12.713,-88.781,168.573,41.435,157.746
C06931=1033.534,12.428,-88.763,168.570,41.436,157.746
C06932=1033.526,12.143,-88.745,168.567,41.437,157.746
C06933=1033.519,11.857,-88.728,168.564,41.438,157.746
C06934=1033.512,11.572,-88.711,168.562,41.439,157.746
C06935=1033.506,11.323,-88.696,168.559,41.439,157.746
C06936=1033.499,11.074,-88.680,168.557,41.440,157.746
C06937=1033.493,10.824,-88.666,168.554,41.441,157.746
C06938=1033.486,10.574,-88.651,168.552,41.442,157.746
C06939=1033.480,10.325,-88.635,168.549,41.442,157.746
C06940=1033.473,10.076,-88.620,168.548,41.443,157.746
C06941=1033.467,9.826,-88.605,168.546,41.444,157.746
C06942=1033.461,9.576,-88.590,168.543,41.444,157.746
C06943=1033.454,9.327,-88.574,168.541,41.445,157.746
C06944=1033.448,9.078,-88.559,168.538,41.446,157.746
C06945=1033.441,8.828,-88.545,168.536,41.447,157.746
C06946=1033.435,8.578,-88.530,168.533,41.448,157.746
C06947=1033.429,8.330,-88.514,168.531,41.449,157.746
C06948=1033.422,8.080,-88.499,168.529,41.449,157.746
C06949=1033.416,7.831,-88.484,168.526,41.450,157.746
C06950=1033.410,7.581,-88.469,168.524,41.451,157.746
C06951=1033.404,7.331,-88.454,168.521,41.451,157.746
C06952=1033.397,7.082,-88.438,168.519,41.452,157.746
C06953=1033.391,6.832,-88.423,168.518,41.453,157.746
C06954=1033.384,6.583,-88.408,168.515,41.453,157.746
C06955=1033.379,6.334,-88.394,168.513,41.454,157.746
C06956=1033.372,6.084,-88.379,168.510,41.455,157.746
C06957=1033.366,5.835,-88.364,168.508,41.456,157.746
C06958=1033.359,5.585,-88.348,168.505,41.457,157.746
C06959=1033.353,5.336,-88.333,168.503,41.458,157.746
C06960=1033.346,5.086,-88.318,168.501,41.458,157.746
C06961=1033.340,4.837,-88.303,168.498,41.459,157.746
C06962=1033.334,4.588,-88.289,168.496,41.460,157.746
C06963=1033.328,4.338,-88.274,168.493,41.460,157.746
C06964=1033.322,4.088,-88.259,168.491,41.461,157.746
C06965=1033.315,3.839,-88.244,168.489,41.462,157.746
C06966=1033.309,3.589,-88.229,168.486,41.462,157.746
C06967=1033.303,3.340,-88.214,168.485,41.463,157.746
C06968=1033.296,3.091,-88.199,168.482,41.464,157.746
C06969=1033.290,2.841,-88.184,168.480,41.465,157.746
C06970=1033.284,2.592,-88.169,168.477,41.466,157.746
C06971=1033.277,2.342,-88.154,168.475,41.466,157.746
C06972=1033.271,2.093,-88.139,168.472,41.467,157.746
C06973=1033.265,1.843,-88.124,168.470,41.468,157.746
C06974=1033.259,1.594,-88.109,168.467,41.468,157.746
C06975=1033.252,1.344,-88.095,168.465,41.469,157.746
C06976=1033.246,1.095,-88.080,168.463,41.469,157.746
C06977=1033.240,0.845,-88.065,168.460,41.470,157.746
C06978=1033.234,0.596,-88.050,168.458,41.471,157.746
C06979=1033.227,0.346,-88.035,168.455,41.472,157.746
C06980=1033.221,0.097,-88.021,168.454,41.473,157.746
C06981=1033.215,-0.153,-88.006,168.450,41.473,157.746
C06982=1033.209,-0.402,-87.991,168.449,41.474,157.746
C06983=1033.202,-0.652,-87.976,168.447,41.475,157.746
C06984=1033.197,-0.901,-87.961,168.444,41.475,157.746
C06985=1033.190,-1.150,-87.946,168.442,41.476,157.746
C06986=1033.184,-1.401,-87.932,168.439,41.477,157.746
C06987=1033.178,-1.650,-87.917,168.437,41.477,157.746
C06988=1033.172,-1.899,-87.902,168.434,41.479,157.746
C06989=1033.166,-2.149,-87.887,168.432,41.479,157.746
C06990=1033.160,-2.398,-87.873,168.430,41.480,157.746
C06991=1033.153,-2.648,-87.858,168.427,41.480,157.746
C06992=1033.147,-2.897,-87.843,168.425,41.481,157.746
C06993=1033.141,-3.146,-87.828,168.422,41.482,157.746
C06994=1033.135,-3.396,-87.813,168.420,41.482,157.746
C06995=1033.128,-3.679,-87.797,168.418,41.483,157.746
C06996=1033.121,-3.963,-87.781,168.415,41.484,157.746
C06997=1033.113,-4.246,-87.764,168.412,41.485,157.746
C06998=1033.105,-4.529,-87.748,168.409,41.486,157.746
C06999=1033.099,-4.778,-87.733,168.407,41.487,157.746
C07000=1033.094,-5.028,-87.719,168.404,41.488,157.746
C07001=1033.086,-5.277,-87.705,168.402,41.489,157.746
C07002=1033.080,-5.527,-87.690,168.399,41.490,157.746
C07003=1033.075,-5.777,-87.676,168.397,41.490,157.746
C07004=1033.068,-6.026,-87.662,168.394,41.491,157.746
C07005=1033.061,-6.276,-87.647,168.392,41.492,157.746
C07006=1033.056,-6.525,-87.633,168.390,41.493,157.746
C07007=1033.049,-6.775,-87.618,168.388,41.494,157.746
C07008=1033.042,-7.024,-87.604,168.385,41.494,157.746
C07009=1033.036,-7.273,-87.590,168.383,41.495,157.746
C07010=1033.030,-7.523,-87.575,168.380,41.496,157.746
C07011=1033.023,-7.773,-87.560,168.378,41.497,157.746
C07012=1033.017,-8.022,-87.547,168.375,41.498,157.746
C07013=1033.011,-8.272,-87.532,168.373,41.498,157.746
C07014=1033.004,-8.521,-87.517,168.370,41.500,157.746
C07015=1032.998,-8.771,-87.504,168.368,41.500,157.746
C07016=1032.992,-9.020,-87.489,168.365,41.501,157.746
C07017=1032.986,-9.269,-87.474,168.364,41.502,157.746
C07018=1032.979,-9.519,-87.461,168.361,41.503,157.746
C07019=1032.973,-9.769,-87.446,168.359,41.504,157.746
C07020=1032.966,-10.018,-87.433,168.356,41.505,157.746
C07021=1032.960,-10.268,-87.418,168.354,41.505,157.746
C07022=1032.955,-10.517,-87.404,168.351,41.506,157.746
C07023=1032.947,-10.767,-87.389,168.349,41.507,157.746
C07024=1032.942,-11.016,-87.376,168.346,41.508,157.746
C07025=1032.935,-11.266,-87.361,168.343,41.508,157.746
C07026=1032.928,-11.515,-87.346,168.341,41.509,157.746
C07027=1032.923,-11.765,-87.332,168.339,41.510,157.746
C07028=1032.916,-12.014,-87.318,168.336,41.511,157.746
C07029=1032.910,-12.264,-87.304,168.334,41.512,157.746
C07030=1032.904,-12.513,-87.289,168.332,41.513,157.746
C07031=1032.898,-12.763,-87.276,168.329,41.514,157.746
C07032=1032.891,-13.012,-87.261,168.327,41.514,157.746
C07033=1032.885,-13.262,-87.248,168.324,41.515,157.746
C07034=1032.879,-13.511,-87.233,168.322,41.516,157.746
C07035=1032.873,-13.761,-87.219,168.319,41.517,157.746
C07036=1032.866,-14.011,-87.205,168.317,41.517,157.746
C07037=1032.861,-14.260,-87.191,168.314,41.518,157.746
C07038=1032.854,-14.510,-87.177,168.312,41.519,157.746
C07039=1032.848,-14.759,-87.162,168.309,41.520,157.746
C07040=1032.842,-15.009,-87.148,168.308,41.520,157.746
C07041=1032.835,-15.258,-87.134,168.305,41.522,157.746
C07042=1032.829,-15.508,-87.120,168.302,41.523,157.746
C07043=1032.823,-15.758,-87.106,168.300,41.523,157.746
C07044=1032.816,-16.006,-87.092,168.297,41.524,157.746
C07045=1032.810,-16.257,-87.078,168.295,41.525,157.746
C07046=1032.804,-16.506,-87.065,168.292,41.526,157.746
C07047=1032.797,-16.755,-87.051,168.290,41.527,157.746
C07048=1032.791,-17.005,-87.037,168.287,41.528,157.746
C07049=1032.784,-17.255,-87.023,168.285,41.529,157.746
C07050=1032.779,-17.505,-87.009,168.283,41.530,157.747
C07051=1032.772,-17.754,-86.995,168.280,41.531,157.747
C07052=1032.766,-18.003,-86.982,168.278,41.531,157.746
C07053=1032.760,-18.253,-86.967,168.275,41.532,157.747
C07054=1032.753,-18.503,-86.954,168.272,41.533,157.747
C07055=1032.747,-18.751,-86.940,168.270,41.534,157.747
C07056=1032.741,-19.002,-86.926,168.267,41.535,157.747
C07057=1032.734,-19.251,-86.913,168.265,41.536,157.747
C07058=1032.728,-19.501,-86.899,168.263,41.537,157.747
C07059=1032.721,-19.782,-86.883,168.260,41.538,157.747
C07060=1032.713,-20.064,-86.867,168.257,41.539,157.747
C07061=1032.707,-20.345,-86.852,168.254,41.540,157.747
C07062=1032.700,-20.627,-86.836,168.251,41.541,157.747
C07063=1032.693,-20.877,-86.823,168.249,41.542,157.747
C07064=1032.687,-21.126,-86.809,168.246,41.543,157.747
C07065=1032.681,-21.376,-86.795,168.243,41.544,157.747
C07066=1032.674,-21.625,-86.782,168.241,41.545,157.747
C07067=1032.668,-21.875,-86.769,168.239,41.546,157.747
C07068=1032.662,-22.124,-86.754,168.237,41.547,157.747
C07069=1032.656,-22.374,-86.740,168.234,41.547,157.747
C07070=1032.649,-22.624,-86.727,168.231,41.548,157.747
C07071=1032.643,-22.873,-86.713,168.229,41.549,157.747
C07072=1032.637,-23.122,-86.700,168.226,41.550,157.747
C07073=1032.630,-23.372,-86.686,168.224,41.551,157.747
C07074=1032.625,-23.622,-86.672,168.221,41.552,157.747
C07075=1032.619,-23.871,-86.659,168.218,41.552,157.747
C07076=1032.612,-24.121,-86.645,168.216,41.553,157.747
C07077=1032.606,-24.370,-86.631,168.214,41.554,157.747
C07078=1032.600,-24.619,-86.617,168.212,41.555,157.747
C07079=1032.593,-24.869,-86.604,168.209,41.556,157.747
C07080=1032.587,-25.119,-86.591,168.206,41.557,157.747
C07081=1032.581,-25.368,-86.577,168.204,41.558,157.747
C07082=1032.574,-25.618,-86.563,168.201,41.559,157.747
C07083=1032.568,-25.867,-86.550,168.199,41.560,157.747
C07084=1032.563,-26.117,-86.536,168.196,41.561,157.747
C07085=1032.556,-26.367,-86.522,168.193,41.562,157.747
C07086=1032.550,-26.616,-86.509,168.191,41.562,157.747
C07087=1032.543,-26.865,-86.496,168.189,41.563,157.747
C07088=1032.538,-27.115,-86.482,168.187,41.564,157.747
C07089=1032.531,-27.365,-86.468,168.184,41.565,157.747
C07090=1032.525,-27.615,-86.456,168.181,41.566,157.747
C07091=1032.519,-27.864,-86.442,168.179,41.567,157.747
C07092=1032.512,-28.114,-86.429,168.176,41.568,157.747
C07093=1032.506,-28.363,-86.415,168.173,41.569,157.747
C07094=1032.500,-28.613,-86.402,168.171,41.570,157.747
C07095=1032.493,-28.863,-86.389,168.169,41.571,157.747
C07096=1032.487,-29.112,-86.375,168.166,41.572,157.747
C07097=1032.481,-29.361,-86.362,168.164,41.573,157.747
C07098=1032.475,-29.611,-86.349,168.161,41.574,157.747
C07099=1032.468,-29.861,-86.336,168.158,41.575,157.747
C07100=1032.462,-30.110,-86.323,168.155,41.576,157.748
C07101=1032.455,-30.359,-86.309,168.153,41.577,157.748
C07102=1032.449,-30.609,-86.296,168.150,41.578,157.748
C07103=1032.443,-30.859,-86.283,168.148,41.579,157.748
C07104=1032.436,-31.109,-86.270,168.146,41.580,157.748
C07105=1032.430,-31.358,-86.257,168.143,41.581,157.748
C07106=1032.424,-31.607,-86.243,168.140,41.582,157.748
C07107=1032.417,-31.857,-86.230,168.138,41.583,157.748
C07108=1032.411,-32.107,-86.217,168.135,41.584,157.748
C07109=1032.405,-32.356,-86.204,168.132,41.585,157.748
C07110=1032.399,-32.605,-86.191,168.130,41.586,157.748
C07111=1032.393,-32.855,-86.178,168.127,41.587,157.748
C07112=1032.386,-33.105,-86.164,168.125,41.588,157.748
C07113=1032.380,-33.355,-86.151,168.123,41.589,157.748
C07114=1032.374,-33.604,-86.138,168.120,41.590,157.748
C07115=1032.368,-33.854,-86.125,168.117,41.591,157.748
C07116=1032.362,-34.103,-86.112,168.115,41.592,157.748
C07117=1032.355,-34.353,-86.098,168.112,41.593,157.748
C07118=1032.349,-34.603,-86.086,168.109,41.594,157.748
C07119=1032.343,-34.852,-86.073,168.107,41.595,157.748
C07120=1032.336,-35.101,-86.059,168.105,41.596,157.748
C07121=1032.331,-35.351,-86.047,168.102,41.597,157.748
C07122=1032.324,-35.601,-86.033,168.099,41.598,157.748
C07123=1032.319,-35.819,-86.022,168.097,41.599,157.748
C07124=1032.314,-36.037,-86.010,168.095,41.599,157.748
C07125=1032.308,-36.255,-85.999,168.092,41.600,157.748
C07126=1032.303,-36.473,-85.987,168.090,41.601,157.748
C07127=1032.297,-36.692,-85.976,168.088,41.602,157.748
C07128=1032.292,-36.909,-85.965,168.085,41.603,157.748
C07129=1032.287,-37.128,-85.953,168.083,41.603,157.748
C07130=1032.281,-37.347,-85.942,168.082,41.604,157.748
C07131=1032.273,-37.690,-85.924,168.078,41.606,157.748
C07132=1032.264,-38.033,-85.907,168.074,41.607,157.748
C07133=1032.256,-38.376,-85.888,168.071,41.608,157.748
C07134=1032.247,-38.721,-85.871,168.067,41.609,157.748
C07135=1032.241,-38.970,-85.858,168.064,41.611,157.748
C07136=1032.235,-39.220,-85.845,168.061,41.612,157.748
C07137=1032.229,-39.470,-85.832,168.060,41.613,157.749
C07138=1032.222,-39.719,-85.820,168.057,41.614,157.749
C07139=1032.216,-39.968,-85.806,168.054,41.615,157.749
C07140=1032.210,-40.218,-85.794,168.051,41.616,157.749
C07141=1032.204,-40.468,-85.781,168.049,41.617,157.749
C07142=1032.197,-40.717,-85.769,168.046,41.618,157.749
C07143=1032.191,-40.968,-85.756,168.044,41.619,157.749
C07144=1032.184,-41.217,-85.743,168.041,41.620,157.749
C07145=1032.179,-41.467,-85.730,168.039,41.621,157.749
C07146=1032.172,-41.716,-85.718,168.036,41.622,157.749
C07147=1032.166,-41.966,-85.705,168.033,41.623,157.749
C07148=1032.160,-42.216,-85.692,168.030,41.625,157.749
C07149=1032.153,-42.465,-85.679,168.028,41.626,157.749
C07150=1032.147,-42.714,-85.667,168.026,41.627,157.749
C07151=1032.141,-42.964,-85.654,168.023,41.628,157.749
C07152=1032.135,-43.214,-85.641,168.020,41.629,157.749
C07153=1032.128,-43.463,-85.629,168.018,41.630,157.749
C07154=1032.122,-43.713,-85.617,168.015,41.631,157.749
C07155=1032.116,-43.963,-85.604,168.012,41.632,157.749
C07156=1032.109,-44.212,-85.591,168.009,41.633,157.749
C07157=1032.103,-44.462,-85.579,168.006,41.634,157.749
C07158=1032.098,-44.712,-85.566,168.005,41.635,157.749
C07159=1032.091,-44.961,-85.554,168.002,41.636,157.749
C07160=1032.085,-45.210,-85.541,167.999,41.638,157.749
C07161=1032.079,-45.460,-85.528,167.996,41.639,157.749
C07162=1032.073,-45.710,-85.516,167.994,41.640,157.750
C07163=1032.066,-45.959,-85.503,167.991,41.641,157.750
C07164=1032.060,-46.209,-85.491,167.989,41.642,157.750
C07165=1032.054,-46.459,-85.478,167.986,41.643,157.750
C07166=1032.047,-46.709,-85.466,167.984,41.644,157.750
C07167=1032.041,-46.958,-85.453,167.981,41.645,157.750
C07168=1032.036,-47.207,-85.441,167.978,41.646,157.750
C07169=1032.029,-47.457,-85.429,167.975,41.647,157.750
C07170=1032.023,-47.706,-85.416,167.972,41.649,157.750
C07171=1032.017,-47.956,-85.404,167.970,41.649,157.750
C07172=1032.011,-48.206,-85.392,167.968,41.651,157.750
C07173=1032.005,-48.455,-85.378,167.965,41.652,157.750
C07174=1031.999,-48.705,-85.366,167.962,41.653,157.750
C07175=1031.992,-48.955,-85.354,167.960,41.654,157.750
C07176=1031.986,-49.204,-85.341,167.957,41.655,157.750
C07177=1031.980,-49.454,-85.329,167.954,41.656,157.750
C07178=1031.974,-49.703,-85.317,167.951,41.657,157.750
C07179=1031.968,-49.953,-85.305,167.950,41.658,157.750
C07180=1031.962,-50.203,-85.292,167.947,41.659,157.750
C07181=1031.956,-50.452,-85.279,167.944,41.661,157.750
C07182=1031.950,-50.702,-85.267,167.941,41.662,157.750
C07183=1031.943,-50.951,-85.255,167.938,41.663,157.750
C07184=1031.937,-51.201,-85.242,167.935,41.664,157.750
C07185=1031.931,-51.451,-85.231,167.934,41.665,157.750
C07186=1031.924,-51.701,-85.219,167.931,41.666,157.750
C07187=1031.917,-51.982,-85.205,167.927,41.668,157.751
C07188=1031.910,-52.264,-85.191,167.924,41.669,157.751
C07189=1031.903,-52.544,-85.178,167.921,41.671,157.751
C07190=1031.896,-52.826,-85.164,167.919,41.672,157.751
C07191=1031.890,-53.075,-85.153,167.916,41.673,157.751
C07192=1031.883,-53.325,-85.141,167.913,41.675,157.751
C07193=1031.877,-53.575,-85.128,167.910,41.676,157.751
C07194=1031.870,-53.824,-85.116,167.907,41.677,157.751
C07195=1031.864,-54.074,-85.104,167.904,41.679,157.751
C07196=1031.858,-54.324,-85.092,167.903,41.680,157.751
C07197=1031.852,-54.573,-85.081,167.900,41.681,157.751
C07198=1031.845,-54.823,-85.069,167.897,41.682,157.751
C07199=1031.840,-55.073,-85.056,167.894,41.684,157.751
C07200=1031.833,-55.322,-85.044,167.891,41.685,157.751
C07201=1031.826,-55.572,-85.032,167.888,41.686,157.751
C07202=1031.820,-55.821,-85.020,167.886,41.687,157.751
C07203=1031.815,-56.071,-85.009,167.883,41.688,157.751
C07204=1031.808,-56.321,-84.997,167.881,41.689,157.752
C07205=1031.801,-56.570,-84.985,167.878,41.690,157.752
C07206=1031.795,-56.820,-84.973,167.875,41.692,157.752
